   STATUS[148].EXT.Operation := FALSE;
   STATUS[148].EXT.Forced := FALSE;
   STATUS[148].EXT.BIT29 := FALSE;
   STATUS[148].EXT.BIT30 := FALSE;
   STATUS[148].EXT.BIT31 := FALSE;
   STATUS[148].EXT.ModeBit1 := FALSE;
   STATUS[148].EXT.ModeBit2 := FALSE;
   STATUS[148].EXT.ModeBit3 := FALSE;
   STATUS[148].EXT.BIT19 := FALSE;
   STATUS[148].EXT.BIT20 := FALSE;
   STATUS[148].EXT.AlarmSuppressed := FALSE;
   STATUS[148].EXT.AlarmPresent := FALSE;
   STATUS[148].EXT.AlarmFailUnAck := FALSE;
   STATUS[148].Status := 0;
   STATUS[148].TimeStamp := 16#0000;
   STATUS[149].EXT.AlarmWarnUnAck := FALSE;
   STATUS[149].EXT.AckRequired := FALSE;
   STATUS[149].EXT.Maintanence := FALSE;
   STATUS[149].EXT.Operation := FALSE;
   STATUS[149].EXT.Forced := FALSE;
   STATUS[149].EXT.BIT29 := FALSE;
   STATUS[149].EXT.BIT30 := FALSE;
   STATUS[149].EXT.BIT31 := FALSE;
   STATUS[149].EXT.ModeBit1 := FALSE;
   STATUS[149].EXT.ModeBit2 := FALSE;
   STATUS[149].EXT.ModeBit3 := FALSE;
   STATUS[149].EXT.BIT19 := FALSE;
   STATUS[149].EXT.BIT20 := FALSE;
   STATUS[149].EXT.AlarmSuppressed := FALSE;
   STATUS[149].EXT.AlarmPresent := FALSE;
   STATUS[149].EXT.AlarmFailUnAck := FALSE;
   STATUS[149].Status := 0;
   STATUS[149].TimeStamp := 16#0000;
   STATUS[150].EXT.AlarmWarnUnAck := FALSE;
   STATUS[150].EXT.AckRequired := FALSE;
   STATUS[150].EXT.Maintanence := FALSE;
   STATUS[150].EXT.Operation := FALSE;
   STATUS[150].EXT.Forced := FALSE;
   STATUS[150].EXT.BIT29 := FALSE;
   STATUS[150].EXT.BIT30 := FALSE;
   STATUS[150].EXT.BIT31 := FALSE;
   STATUS[150].EXT.ModeBit1 := FALSE;
   STATUS[150].EXT.ModeBit2 := FALSE;
   STATUS[150].EXT.ModeBit3 := FALSE;
   STATUS[150].EXT.BIT19 := FALSE;
   STATUS[150].EXT.BIT20 := FALSE;
   STATUS[150].EXT.AlarmSuppressed := FALSE;
   STATUS[150].EXT.AlarmPresent := FALSE;
   STATUS[150].EXT.AlarmFailUnAck := FALSE;
   STATUS[150].Status := 0;
   STATUS[150].TimeStamp := 16#0000;
   STATUS[151].EXT.AlarmWarnUnAck := FALSE;
   STATUS[151].EXT.AckRequired := FALSE;
   STATUS[151].EXT.Maintanence := FALSE;
   STATUS[151].EXT.Operation := FALSE;
   STATUS[151].EXT.Forced := FALSE;
   STATUS[151].EXT.BIT29 := FALSE;
   STATUS[151].EXT.BIT30 := FALSE;
   STATUS[151].EXT.BIT31 := FALSE;
   STATUS[151].EXT.ModeBit1 := FALSE;
   STATUS[151].EXT.ModeBit2 := FALSE;
   STATUS[151].EXT.ModeBit3 := FALSE;
   STATUS[151].EXT.BIT19 := FALSE;
   STATUS[151].EXT.BIT20 := FALSE;
   STATUS[151].EXT.AlarmSuppressed := FALSE;
   STATUS[151].EXT.AlarmPresent := FALSE;
   STATUS[151].EXT.AlarmFailUnAck := FALSE;
   STATUS[151].Status := 0;
   STATUS[151].TimeStamp := 16#0000;
   STATUS[152].EXT.AlarmWarnUnAck := FALSE;
   STATUS[152].EXT.AckRequired := FALSE;
   STATUS[152].EXT.Maintanence := FALSE;
   STATUS[152].EXT.Operation := FALSE;
   STATUS[152].EXT.Forced := FALSE;
   STATUS[152].EXT.BIT29 := FALSE;
   STATUS[152].EXT.BIT30 := FALSE;
   STATUS[152].EXT.BIT31 := FALSE;
   STATUS[152].EXT.ModeBit1 := FALSE;
   STATUS[152].EXT.ModeBit2 := FALSE;
   STATUS[152].EXT.ModeBit3 := FALSE;
   STATUS[152].EXT.BIT19 := FALSE;
   STATUS[152].EXT.BIT20 := FALSE;
   STATUS[152].EXT.AlarmSuppressed := FALSE;
   STATUS[152].EXT.AlarmPresent := FALSE;
   STATUS[152].EXT.AlarmFailUnAck := FALSE;
   STATUS[152].Status := 0;
   STATUS[152].TimeStamp := 16#0000;
   STATUS[153].EXT.AlarmWarnUnAck := FALSE;
   STATUS[153].EXT.AckRequired := FALSE;
   STATUS[153].EXT.Maintanence := FALSE;
   STATUS[153].EXT.Operation := FALSE;
   STATUS[153].EXT.Forced := FALSE;
   STATUS[153].EXT.BIT29 := FALSE;
   STATUS[153].EXT.BIT30 := FALSE;
   STATUS[153].EXT.BIT31 := FALSE;
   STATUS[153].EXT.ModeBit1 := FALSE;
   STATUS[153].EXT.ModeBit2 := FALSE;
   STATUS[153].EXT.ModeBit3 := FALSE;
   STATUS[153].EXT.BIT19 := FALSE;
   STATUS[153].EXT.BIT20 := FALSE;
   STATUS[153].EXT.AlarmSuppressed := FALSE;
   STATUS[153].EXT.AlarmPresent := FALSE;
   STATUS[153].EXT.AlarmFailUnAck := FALSE;
   STATUS[153].Status := 0;
   STATUS[153].TimeStamp := 16#0000;
   STATUS[154].EXT.AlarmWarnUnAck := FALSE;
   STATUS[154].EXT.AckRequired := FALSE;
   STATUS[154].EXT.Maintanence := FALSE;
   STATUS[154].EXT.Operation := FALSE;
   STATUS[154].EXT.Forced := FALSE;
   STATUS[154].EXT.BIT29 := FALSE;
   STATUS[154].EXT.BIT30 := FALSE;
   STATUS[154].EXT.BIT31 := FALSE;
   STATUS[154].EXT.ModeBit1 := FALSE;
   STATUS[154].EXT.ModeBit2 := FALSE;
   STATUS[154].EXT.ModeBit3 := FALSE;
   STATUS[154].EXT.BIT19 := FALSE;
   STATUS[154].EXT.BIT20 := FALSE;
   STATUS[154].EXT.AlarmSuppressed := FALSE;
   STATUS[154].EXT.AlarmPresent := FALSE;
   STATUS[154].EXT.AlarmFailUnAck := FALSE;
   STATUS[154].Status := 0;
   STATUS[154].TimeStamp := 16#0000;
   STATUS[155].EXT.AlarmWarnUnAck := FALSE;
   STATUS[155].EXT.AckRequired := FALSE;
   STATUS[155].EXT.Maintanence := FALSE;
   STATUS[155].EXT.Operation := FALSE;
   STATUS[155].EXT.Forced := FALSE;
   STATUS[155].EXT.BIT29 := FALSE;
   STATUS[155].EXT.BIT30 := FALSE;
   STATUS[155].EXT.BIT31 := FALSE;
   STATUS[155].EXT.ModeBit1 := FALSE;
   STATUS[155].EXT.ModeBit2 := FALSE;
   STATUS[155].EXT.ModeBit3 := FALSE;
   STATUS[155].EXT.BIT19 := FALSE;
   STATUS[155].EXT.BIT20 := FALSE;
   STATUS[155].EXT.AlarmSuppressed := FALSE;
   STATUS[155].EXT.AlarmPresent := FALSE;
   STATUS[155].EXT.AlarmFailUnAck := FALSE;
   STATUS[155].Status := 0;
   STATUS[155].TimeStamp := 16#0000;
   STATUS[156].EXT.AlarmWarnUnAck := FALSE;
   STATUS[156].EXT.AckRequired := FALSE;
   STATUS[156].EXT.Maintanence := FALSE;
   STATUS[156].EXT.Operation := FALSE;
   STATUS[156].EXT.Forced := FALSE;
   STATUS[156].EXT.BIT29 := FALSE;
   STATUS[156].EXT.BIT30 := FALSE;
   STATUS[156].EXT.BIT31 := FALSE;
   STATUS[156].EXT.ModeBit1 := FALSE;
   STATUS[156].EXT.ModeBit2 := FALSE;
   STATUS[156].EXT.ModeBit3 := FALSE;
   STATUS[156].EXT.BIT19 := FALSE;
   STATUS[156].EXT.BIT20 := FALSE;
   STATUS[156].EXT.AlarmSuppressed := FALSE;
   STATUS[156].EXT.AlarmPresent := FALSE;
   STATUS[156].EXT.AlarmFailUnAck := FALSE;
   STATUS[156].Status := 0;
   STATUS[156].TimeStamp := 16#0000;
   STATUS[157].EXT.AlarmWarnUnAck := FALSE;
   STATUS[157].EXT.AckRequired := FALSE;
   STATUS[157].EXT.Maintanence := FALSE;
   STATUS[157].EXT.Operation := FALSE;
   STATUS[157].EXT.Forced := FALSE;
   STATUS[157].EXT.BIT29 := FALSE;
   STATUS[157].EXT.BIT30 := FALSE;
   STATUS[157].EXT.BIT31 := FALSE;
   STATUS[157].EXT.ModeBit1 := FALSE;
   STATUS[157].EXT.ModeBit2 := FALSE;
   STATUS[157].EXT.ModeBit3 := FALSE;
   STATUS[157].EXT.BIT19 := FALSE;
   STATUS[157].EXT.BIT20 := FALSE;
   STATUS[157].EXT.AlarmSuppressed := FALSE;
   STATUS[157].EXT.AlarmPresent := FALSE;
   STATUS[157].EXT.AlarmFailUnAck := FALSE;
   STATUS[157].Status := 0;
   STATUS[157].TimeStamp := 16#0000;
   STATUS[158].EXT.AlarmWarnUnAck := FALSE;
   STATUS[158].EXT.AckRequired := FALSE;
   STATUS[158].EXT.Maintanence := FALSE;
   STATUS[158].EXT.Operation := FALSE;
   STATUS[158].EXT.Forced := FALSE;
   STATUS[158].EXT.BIT29 := FALSE;
   STATUS[158].EXT.BIT30 := FALSE;
   STATUS[158].EXT.BIT31 := FALSE;
   STATUS[158].EXT.ModeBit1 := FALSE;
   STATUS[158].EXT.ModeBit2 := FALSE;
   STATUS[158].EXT.ModeBit3 := FALSE;
   STATUS[158].EXT.BIT19 := FALSE;
   STATUS[158].EXT.BIT20 := FALSE;
   STATUS[158].EXT.AlarmSuppressed := FALSE;
   STATUS[158].EXT.AlarmPresent := FALSE;
   STATUS[158].EXT.AlarmFailUnAck := FALSE;
   STATUS[158].Status := 0;
   STATUS[158].TimeStamp := 16#0000;
   STATUS[159].EXT.AlarmWarnUnAck := FALSE;
   STATUS[159].EXT.AckRequired := FALSE;
   STATUS[159].EXT.Maintanence := FALSE;
   STATUS[159].EXT.Operation := FALSE;
   STATUS[159].EXT.Forced := FALSE;
   STATUS[159].EXT.BIT29 := FALSE;
   STATUS[159].EXT.BIT30 := FALSE;
   STATUS[159].EXT.BIT31 := FALSE;
   STATUS[159].EXT.ModeBit1 := FALSE;
   STATUS[159].EXT.ModeBit2 := FALSE;
   STATUS[159].EXT.ModeBit3 := FALSE;
   STATUS[159].EXT.BIT19 := FALSE;
   STATUS[159].EXT.BIT20 := FALSE;
   STATUS[159].EXT.AlarmSuppressed := FALSE;
   STATUS[159].EXT.AlarmPresent := FALSE;
   STATUS[159].EXT.AlarmFailUnAck := FALSE;
   STATUS[159].Status := 0;
   STATUS[159].TimeStamp := 16#0000;
   STATUS[160].EXT.AlarmWarnUnAck := FALSE;
   STATUS[160].EXT.AckRequired := FALSE;
   STATUS[160].EXT.Maintanence := FALSE;
   STATUS[160].EXT.Operation := FALSE;
   STATUS[160].EXT.Forced := FALSE;
   STATUS[160].EXT.BIT29 := FALSE;
   STATUS[160].EXT.BIT30 := FALSE;
   STATUS[160].EXT.BIT31 := FALSE;
   STATUS[160].EXT.ModeBit1 := FALSE;
   STATUS[160].EXT.ModeBit2 := FALSE;
   STATUS[160].EXT.ModeBit3 := FALSE;
   STATUS[160].EXT.BIT19 := FALSE;
   STATUS[160].EXT.BIT20 := FALSE;
   STATUS[160].EXT.AlarmSuppressed := FALSE;
   STATUS[160].EXT.AlarmPresent := FALSE;
   STATUS[160].EXT.AlarmFailUnAck := FALSE;
   STATUS[160].Status := 0;
   STATUS[160].TimeStamp := 16#0000;
   STATUS[161].EXT.AlarmWarnUnAck := FALSE;
   STATUS[161].EXT.AckRequired := FALSE;
   STATUS[161].EXT.Maintanence := FALSE;
   STATUS[161].EXT.Operation := FALSE;
   STATUS[161].EXT.Forced := FALSE;
   STATUS[161].EXT.BIT29 := FALSE;
   STATUS[161].EXT.BIT30 := FALSE;
   STATUS[161].EXT.BIT31 := FALSE;
   STATUS[161].EXT.ModeBit1 := FALSE;
   STATUS[161].EXT.ModeBit2 := FALSE;
   STATUS[161].EXT.ModeBit3 := FALSE;
   STATUS[161].EXT.BIT19 := FALSE;
   STATUS[161].EXT.BIT20 := FALSE;
   STATUS[161].EXT.AlarmSuppressed := FALSE;
   STATUS[161].EXT.AlarmPresent := FALSE;
   STATUS[161].EXT.AlarmFailUnAck := FALSE;
   STATUS[161].Status := 0;
   STATUS[161].TimeStamp := 16#0000;
   STATUS[162].EXT.AlarmWarnUnAck := FALSE;
   STATUS[162].EXT.AckRequired := FALSE;
   STATUS[162].EXT.Maintanence := FALSE;
   STATUS[162].EXT.Operation := FALSE;
   STATUS[162].EXT.Forced := FALSE;
   STATUS[162].EXT.BIT29 := FALSE;
   STATUS[162].EXT.BIT30 := FALSE;
   STATUS[162].EXT.BIT31 := FALSE;
   STATUS[162].EXT.ModeBit1 := FALSE;
   STATUS[162].EXT.ModeBit2 := FALSE;
   STATUS[162].EXT.ModeBit3 := FALSE;
   STATUS[162].EXT.BIT19 := FALSE;
   STATUS[162].EXT.BIT20 := FALSE;
   STATUS[162].EXT.AlarmSuppressed := FALSE;
   STATUS[162].EXT.AlarmPresent := FALSE;
   STATUS[162].EXT.AlarmFailUnAck := FALSE;
   STATUS[162].Status := 0;
   STATUS[162].TimeStamp := 16#0000;
   STATUS[163].EXT.AlarmWarnUnAck := FALSE;
   STATUS[163].EXT.AckRequired := FALSE;
   STATUS[163].EXT.Maintanence := FALSE;
   STATUS[163].EXT.Operation := FALSE;
   STATUS[163].EXT.Forced := FALSE;
   STATUS[163].EXT.BIT29 := FALSE;
   STATUS[163].EXT.BIT30 := FALSE;
   STATUS[163].EXT.BIT31 := FALSE;
   STATUS[163].EXT.ModeBit1 := FALSE;
   STATUS[163].EXT.ModeBit2 := FALSE;
   STATUS[163].EXT.ModeBit3 := FALSE;
   STATUS[163].EXT.BIT19 := FALSE;
   STATUS[163].EXT.BIT20 := FALSE;
   STATUS[163].EXT.AlarmSuppressed := FALSE;
   STATUS[163].EXT.AlarmPresent := FALSE;
   STATUS[163].EXT.AlarmFailUnAck := FALSE;
   STATUS[163].Status := 0;
   STATUS[163].TimeStamp := 16#0000;
   STATUS[164].EXT.AlarmWarnUnAck := FALSE;
   STATUS[164].EXT.AckRequired := FALSE;
   STATUS[164].EXT.Maintanence := FALSE;
   STATUS[164].EXT.Operation := FALSE;
   STATUS[164].EXT.Forced := FALSE;
   STATUS[164].EXT.BIT29 := FALSE;
   STATUS[164].EXT.BIT30 := FALSE;
   STATUS[164].EXT.BIT31 := FALSE;
   STATUS[164].EXT.ModeBit1 := FALSE;
   STATUS[164].EXT.ModeBit2 := FALSE;
   STATUS[164].EXT.ModeBit3 := FALSE;
   STATUS[164].EXT.BIT19 := FALSE;
   STATUS[164].EXT.BIT20 := FALSE;
   STATUS[164].EXT.AlarmSuppressed := FALSE;
   STATUS[164].EXT.AlarmPresent := FALSE;
   STATUS[164].EXT.AlarmFailUnAck := FALSE;
   STATUS[164].Status := 0;
   STATUS[164].TimeStamp := 16#0000;
   STATUS[165].EXT.AlarmWarnUnAck := FALSE;
   STATUS[165].EXT.AckRequired := FALSE;
   STATUS[165].EXT.Maintanence := FALSE;
   STATUS[165].EXT.Operation := FALSE;
   STATUS[165].EXT.Forced := FALSE;
   STATUS[165].EXT.BIT29 := FALSE;
   STATUS[165].EXT.BIT30 := FALSE;
   STATUS[165].EXT.BIT31 := FALSE;
   STATUS[165].EXT.ModeBit1 := FALSE;
   STATUS[165].EXT.ModeBit2 := FALSE;
   STATUS[165].EXT.ModeBit3 := FALSE;
   STATUS[165].EXT.BIT19 := FALSE;
   STATUS[165].EXT.BIT20 := FALSE;
   STATUS[165].EXT.AlarmSuppressed := FALSE;
   STATUS[165].EXT.AlarmPresent := FALSE;
   STATUS[165].EXT.AlarmFailUnAck := FALSE;
   STATUS[165].Status := 0;
   STATUS[165].TimeStamp := 16#0000;
   STATUS[166].EXT.AlarmWarnUnAck := FALSE;
   STATUS[166].EXT.AckRequired := FALSE;
   STATUS[166].EXT.Maintanence := FALSE;
   STATUS[166].EXT.Operation := FALSE;
   STATUS[166].EXT.Forced := FALSE;
   STATUS[166].EXT.BIT29 := FALSE;
   STATUS[166].EXT.BIT30 := FALSE;
   STATUS[166].EXT.BIT31 := FALSE;
   STATUS[166].EXT.ModeBit1 := FALSE;
   STATUS[166].EXT.ModeBit2 := FALSE;
   STATUS[166].EXT.ModeBit3 := FALSE;
   STATUS[166].EXT.BIT19 := FALSE;
   STATUS[166].EXT.BIT20 := FALSE;
   STATUS[166].EXT.AlarmSuppressed := FALSE;
   STATUS[166].EXT.AlarmPresent := FALSE;
   STATUS[166].EXT.AlarmFailUnAck := FALSE;
   STATUS[166].Status := 0;
   STATUS[166].TimeStamp := 16#0000;
   STATUS[167].EXT.AlarmWarnUnAck := FALSE;
   STATUS[167].EXT.AckRequired := FALSE;
   STATUS[167].EXT.Maintanence := FALSE;
   STATUS[167].EXT.Operation := FALSE;
   STATUS[167].EXT.Forced := FALSE;
   STATUS[167].EXT.BIT29 := FALSE;
   STATUS[167].EXT.BIT30 := FALSE;
   STATUS[167].EXT.BIT31 := FALSE;
   STATUS[167].EXT.ModeBit1 := FALSE;
   STATUS[167].EXT.ModeBit2 := FALSE;
   STATUS[167].EXT.ModeBit3 := FALSE;
   STATUS[167].EXT.BIT19 := FALSE;
   STATUS[167].EXT.BIT20 := FALSE;
   STATUS[167].EXT.AlarmSuppressed := FALSE;
   STATUS[167].EXT.AlarmPresent := FALSE;
   STATUS[167].EXT.AlarmFailUnAck := FALSE;
   STATUS[167].Status := 0;
   STATUS[167].TimeStamp := 16#0000;
   STATUS[168].EXT.AlarmWarnUnAck := FALSE;
   STATUS[168].EXT.AckRequired := FALSE;
   STATUS[168].EXT.Maintanence := FALSE;
   STATUS[168].EXT.Operation := FALSE;
   STATUS[168].EXT.Forced := FALSE;
   STATUS[168].EXT.BIT29 := FALSE;
   STATUS[168].EXT.BIT30 := FALSE;
   STATUS[168].EXT.BIT31 := FALSE;
   STATUS[168].EXT.ModeBit1 := FALSE;
   STATUS[168].EXT.ModeBit2 := FALSE;
   STATUS[168].EXT.ModeBit3 := FALSE;
   STATUS[168].EXT.BIT19 := FALSE;
   STATUS[168].EXT.BIT20 := FALSE;
   STATUS[168].EXT.AlarmSuppressed := FALSE;
   STATUS[168].EXT.AlarmPresent := FALSE;
   STATUS[168].EXT.AlarmFailUnAck := FALSE;
   STATUS[168].Status := 0;
   STATUS[168].TimeStamp := 16#0000;
   STATUS[169].EXT.AlarmWarnUnAck := FALSE;
   STATUS[169].EXT.AckRequired := FALSE;
   STATUS[169].EXT.Maintanence := FALSE;
   STATUS[169].EXT.Operation := FALSE;
   STATUS[169].EXT.Forced := FALSE;
   STATUS[169].EXT.BIT29 := FALSE;
   STATUS[169].EXT.BIT30 := FALSE;
   STATUS[169].EXT.BIT31 := FALSE;
   STATUS[169].EXT.ModeBit1 := FALSE;
   STATUS[169].EXT.ModeBit2 := FALSE;
   STATUS[169].EXT.ModeBit3 := FALSE;
   STATUS[169].EXT.BIT19 := FALSE;
   STATUS[169].EXT.BIT20 := FALSE;
   STATUS[169].EXT.AlarmSuppressed := FALSE;
   STATUS[169].EXT.AlarmPresent := FALSE;
   STATUS[169].EXT.AlarmFailUnAck := FALSE;
   STATUS[169].Status := 0;
   STATUS[169].TimeStamp := 16#0000;
   STATUS[170].EXT.AlarmWarnUnAck := FALSE;
   STATUS[170].EXT.AckRequired := FALSE;
   STATUS[170].EXT.Maintanence := FALSE;
   STATUS[170].EXT.Operation := FALSE;
   STATUS[170].EXT.Forced := FALSE;
   STATUS[170].EXT.BIT29 := FALSE;
   STATUS[170].EXT.BIT30 := FALSE;
   STATUS[170].EXT.BIT31 := FALSE;
   STATUS[170].EXT.ModeBit1 := FALSE;
   STATUS[170].EXT.ModeBit2 := FALSE;
   STATUS[170].EXT.ModeBit3 := FALSE;
   STATUS[170].EXT.BIT19 := FALSE;
   STATUS[170].EXT.BIT20 := FALSE;
   STATUS[170].EXT.AlarmSuppressed := FALSE;
   STATUS[170].EXT.AlarmPresent := FALSE;
   STATUS[170].EXT.AlarmFailUnAck := FALSE;
   STATUS[170].Status := 0;
   STATUS[170].TimeStamp := 16#0000;
   STATUS[171].EXT.AlarmWarnUnAck := FALSE;
   STATUS[171].EXT.AckRequired := FALSE;
   STATUS[171].EXT.Maintanence := FALSE;
   STATUS[171].EXT.Operation := FALSE;
   STATUS[171].EXT.Forced := FALSE;
   STATUS[171].EXT.BIT29 := FALSE;
   STATUS[171].EXT.BIT30 := FALSE;
   STATUS[171].EXT.BIT31 := FALSE;
   STATUS[171].EXT.ModeBit1 := FALSE;
   STATUS[171].EXT.ModeBit2 := FALSE;
   STATUS[171].EXT.ModeBit3 := FALSE;
   STATUS[171].EXT.BIT19 := FALSE;
   STATUS[171].EXT.BIT20 := FALSE;
   STATUS[171].EXT.AlarmSuppressed := FALSE;
   STATUS[171].EXT.AlarmPresent := FALSE;
   STATUS[171].EXT.AlarmFailUnAck := FALSE;
   STATUS[171].Status := 0;
   STATUS[171].TimeStamp := 16#0000;
   STATUS[172].EXT.AlarmWarnUnAck := FALSE;
   STATUS[172].EXT.AckRequired := FALSE;
   STATUS[172].EXT.Maintanence := FALSE;
   STATUS[172].EXT.Operation := FALSE;
   STATUS[172].EXT.Forced := FALSE;
   STATUS[172].EXT.BIT29 := FALSE;
   STATUS[172].EXT.BIT30 := FALSE;
   STATUS[172].EXT.BIT31 := FALSE;
   STATUS[172].EXT.ModeBit1 := FALSE;
   STATUS[172].EXT.ModeBit2 := FALSE;
   STATUS[172].EXT.ModeBit3 := FALSE;
   STATUS[172].EXT.BIT19 := FALSE;
   STATUS[172].EXT.BIT20 := FALSE;
   STATUS[172].EXT.AlarmSuppressed := FALSE;
   STATUS[172].EXT.AlarmPresent := FALSE;
   STATUS[172].EXT.AlarmFailUnAck := FALSE;
   STATUS[172].Status := 0;
   STATUS[172].TimeStamp := 16#0000;
   STATUS[173].EXT.AlarmWarnUnAck := FALSE;
   STATUS[173].EXT.AckRequired := FALSE;
   STATUS[173].EXT.Maintanence := FALSE;
   STATUS[173].EXT.Operation := FALSE;
   STATUS[173].EXT.Forced := FALSE;
   STATUS[173].EXT.BIT29 := FALSE;
   STATUS[173].EXT.BIT30 := FALSE;
   STATUS[173].EXT.BIT31 := FALSE;
   STATUS[173].EXT.ModeBit1 := FALSE;
   STATUS[173].EXT.ModeBit2 := FALSE;
   STATUS[173].EXT.ModeBit3 := FALSE;
   STATUS[173].EXT.BIT19 := FALSE;
   STATUS[173].EXT.BIT20 := FALSE;
   STATUS[173].EXT.AlarmSuppressed := FALSE;
   STATUS[173].EXT.AlarmPresent := FALSE;
   STATUS[173].EXT.AlarmFailUnAck := FALSE;
   STATUS[173].Status := 0;
   STATUS[173].TimeStamp := 16#0000;
   STATUS[174].EXT.AlarmWarnUnAck := FALSE;
   STATUS[174].EXT.AckRequired := FALSE;
   STATUS[174].EXT.Maintanence := FALSE;
   STATUS[174].EXT.Operation := FALSE;
   STATUS[174].EXT.Forced := FALSE;
   STATUS[174].EXT.BIT29 := FALSE;
   STATUS[174].EXT.BIT30 := FALSE;
   STATUS[174].EXT.BIT31 := FALSE;
   STATUS[174].EXT.ModeBit1 := FALSE;
   STATUS[174].EXT.ModeBit2 := FALSE;
   STATUS[174].EXT.ModeBit3 := FALSE;
   STATUS[174].EXT.BIT19 := FALSE;
   STATUS[174].EXT.BIT20 := FALSE;
   STATUS[174].EXT.AlarmSuppressed := FALSE;
   STATUS[174].EXT.AlarmPresent := FALSE;
   STATUS[174].EXT.AlarmFailUnAck := FALSE;
   STATUS[174].Status := 0;
   STATUS[174].TimeStamp := 16#0000;
   STATUS[175].EXT.AlarmWarnUnAck := FALSE;
   STATUS[175].EXT.AckRequired := FALSE;
   STATUS[175].EXT.Maintanence := FALSE;
   STATUS[175].EXT.Operation := FALSE;
   STATUS[175].EXT.Forced := FALSE;
   STATUS[175].EXT.BIT29 := FALSE;
   STATUS[175].EXT.BIT30 := FALSE;
   STATUS[175].EXT.BIT31 := FALSE;
   STATUS[175].EXT.ModeBit1 := FALSE;
   STATUS[175].EXT.ModeBit2 := FALSE;
   STATUS[175].EXT.ModeBit3 := FALSE;
   STATUS[175].EXT.BIT19 := FALSE;
   STATUS[175].EXT.BIT20 := FALSE;
   STATUS[175].EXT.AlarmSuppressed := FALSE;
   STATUS[175].EXT.AlarmPresent := FALSE;
   STATUS[175].EXT.AlarmFailUnAck := FALSE;
   STATUS[175].Status := 0;
   STATUS[175].TimeStamp := 16#0000;
   STATUS[176].EXT.AlarmWarnUnAck := FALSE;
   STATUS[176].EXT.AckRequired := FALSE;
   STATUS[176].EXT.Maintanence := FALSE;
   STATUS[176].EXT.Operation := FALSE;
   STATUS[176].EXT.Forced := FALSE;
   STATUS[176].EXT.BIT29 := FALSE;
   STATUS[176].EXT.BIT30 := FALSE;
   STATUS[176].EXT.BIT31 := FALSE;
   STATUS[176].EXT.ModeBit1 := FALSE;
   STATUS[176].EXT.ModeBit2 := FALSE;
   STATUS[176].EXT.ModeBit3 := FALSE;
   STATUS[176].EXT.BIT19 := FALSE;
   STATUS[176].EXT.BIT20 := FALSE;
   STATUS[176].EXT.AlarmSuppressed := FALSE;
   STATUS[176].EXT.AlarmPresent := FALSE;
   STATUS[176].EXT.AlarmFailUnAck := FALSE;
   STATUS[176].Status := 0;
   STATUS[176].TimeStamp := 16#0000;
   STATUS[177].EXT.AlarmWarnUnAck := FALSE;
   STATUS[177].EXT.AckRequired := FALSE;
   STATUS[177].EXT.Maintanence := FALSE;
   STATUS[177].EXT.Operation := FALSE;
   STATUS[177].EXT.Forced := FALSE;
   STATUS[177].EXT.BIT29 := FALSE;
   STATUS[177].EXT.BIT30 := FALSE;
   STATUS[177].EXT.BIT31 := FALSE;
   STATUS[177].EXT.ModeBit1 := FALSE;
   STATUS[177].EXT.ModeBit2 := FALSE;
   STATUS[177].EXT.ModeBit3 := FALSE;
   STATUS[177].EXT.BIT19 := FALSE;
   STATUS[177].EXT.BIT20 := FALSE;
   STATUS[177].EXT.AlarmSuppressed := FALSE;
   STATUS[177].EXT.AlarmPresent := FALSE;
   STATUS[177].EXT.AlarmFailUnAck := FALSE;
   STATUS[177].Status := 0;
   STATUS[177].TimeStamp := 16#0000;
   STATUS[178].EXT.AlarmWarnUnAck := FALSE;
   STATUS[178].EXT.AckRequired := FALSE;
   STATUS[178].EXT.Maintanence := FALSE;
   STATUS[178].EXT.Operation := FALSE;
   STATUS[178].EXT.Forced := FALSE;
   STATUS[178].EXT.BIT29 := FALSE;
   STATUS[178].EXT.BIT30 := FALSE;
   STATUS[178].EXT.BIT31 := FALSE;
   STATUS[178].EXT.ModeBit1 := FALSE;
   STATUS[178].EXT.ModeBit2 := FALSE;
   STATUS[178].EXT.ModeBit3 := FALSE;
   STATUS[178].EXT.BIT19 := FALSE;
   STATUS[178].EXT.BIT20 := FALSE;
   STATUS[178].EXT.AlarmSuppressed := FALSE;
   STATUS[178].EXT.AlarmPresent := FALSE;
   STATUS[178].EXT.AlarmFailUnAck := FALSE;
   STATUS[178].Status := 0;
   STATUS[178].TimeStamp := 16#0000;
   STATUS[179].EXT.AlarmWarnUnAck := FALSE;
   STATUS[179].EXT.AckRequired := FALSE;
   STATUS[179].EXT.Maintanence := FALSE;
   STATUS[179].EXT.Operation := FALSE;
   STATUS[179].EXT.Forced := FALSE;
   STATUS[179].EXT.BIT29 := FALSE;
   STATUS[179].EXT.BIT30 := FALSE;
   STATUS[179].EXT.BIT31 := FALSE;
   STATUS[179].EXT.ModeBit1 := FALSE;
   STATUS[179].EXT.ModeBit2 := FALSE;
   STATUS[179].EXT.ModeBit3 := FALSE;
   STATUS[179].EXT.BIT19 := FALSE;
   STATUS[179].EXT.BIT20 := FALSE;
   STATUS[179].EXT.AlarmSuppressed := FALSE;
   STATUS[179].EXT.AlarmPresent := FALSE;
   STATUS[179].EXT.AlarmFailUnAck := FALSE;
   STATUS[179].Status := 0;
   STATUS[179].TimeStamp := 16#0000;
   STATUS[180].EXT.AlarmWarnUnAck := FALSE;
   STATUS[180].EXT.AckRequired := FALSE;
   STATUS[180].EXT.Maintanence := FALSE;
   STATUS[180].EXT.Operation := FALSE;
   STATUS[180].EXT.Forced := FALSE;
   STATUS[180].EXT.BIT29 := FALSE;
   STATUS[180].EXT.BIT30 := FALSE;
   STATUS[180].EXT.BIT31 := FALSE;
   STATUS[180].EXT.ModeBit1 := FALSE;
   STATUS[180].EXT.ModeBit2 := FALSE;
   STATUS[180].EXT.ModeBit3 := FALSE;
   STATUS[180].EXT.BIT19 := FALSE;
   STATUS[180].EXT.BIT20 := FALSE;
   STATUS[180].EXT.AlarmSuppressed := FALSE;
   STATUS[180].EXT.AlarmPresent := FALSE;
   STATUS[180].EXT.AlarmFailUnAck := FALSE;
   STATUS[180].Status := 0;
   STATUS[180].TimeStamp := 16#0000;
   STATUS[181].EXT.AlarmWarnUnAck := FALSE;
   STATUS[181].EXT.AckRequired := FALSE;
   STATUS[181].EXT.Maintanence := FALSE;
   STATUS[181].EXT.Operation := FALSE;
   STATUS[181].EXT.Forced := FALSE;
   STATUS[181].EXT.BIT29 := FALSE;
   STATUS[181].EXT.BIT30 := FALSE;
   STATUS[181].EXT.BIT31 := FALSE;
   STATUS[181].EXT.ModeBit1 := FALSE;
   STATUS[181].EXT.ModeBit2 := FALSE;
   STATUS[181].EXT.ModeBit3 := FALSE;
   STATUS[181].EXT.BIT19 := FALSE;
   STATUS[181].EXT.BIT20 := FALSE;
   STATUS[181].EXT.AlarmSuppressed := FALSE;
   STATUS[181].EXT.AlarmPresent := FALSE;
   STATUS[181].EXT.AlarmFailUnAck := FALSE;
   STATUS[181].Status := 0;
   STATUS[181].TimeStamp := 16#0000;
   STATUS[182].EXT.AlarmWarnUnAck := FALSE;
   STATUS[182].EXT.AckRequired := FALSE;
   STATUS[182].EXT.Maintanence := FALSE;
   STATUS[182].EXT.Operation := FALSE;
   STATUS[182].EXT.Forced := FALSE;
   STATUS[182].EXT.BIT29 := FALSE;
   STATUS[182].EXT.BIT30 := FALSE;
   STATUS[182].EXT.BIT31 := FALSE;
   STATUS[182].EXT.ModeBit1 := FALSE;
   STATUS[182].EXT.ModeBit2 := FALSE;
   STATUS[182].EXT.ModeBit3 := FALSE;
   STATUS[182].EXT.BIT19 := FALSE;
   STATUS[182].EXT.BIT20 := FALSE;
   STATUS[182].EXT.AlarmSuppressed := FALSE;
   STATUS[182].EXT.AlarmPresent := FALSE;
   STATUS[182].EXT.AlarmFailUnAck := FALSE;
   STATUS[182].Status := 0;
   STATUS[182].TimeStamp := 16#0000;
   STATUS[183].EXT.AlarmWarnUnAck := FALSE;
   STATUS[183].EXT.AckRequired := FALSE;
   STATUS[183].EXT.Maintanence := FALSE;
   STATUS[183].EXT.Operation := FALSE;
   STATUS[183].EXT.Forced := FALSE;
   STATUS[183].EXT.BIT29 := FALSE;
   STATUS[183].EXT.BIT30 := FALSE;
   STATUS[183].EXT.BIT31 := FALSE;
   STATUS[183].EXT.ModeBit1 := FALSE;
   STATUS[183].EXT.ModeBit2 := FALSE;
   STATUS[183].EXT.ModeBit3 := FALSE;
   STATUS[183].EXT.BIT19 := FALSE;
   STATUS[183].EXT.BIT20 := FALSE;
   STATUS[183].EXT.AlarmSuppressed := FALSE;
   STATUS[183].EXT.AlarmPresent := FALSE;
   STATUS[183].EXT.AlarmFailUnAck := FALSE;
   STATUS[183].Status := 0;
   STATUS[183].TimeStamp := 16#0000;
   STATUS[184].EXT.AlarmWarnUnAck := FALSE;
   STATUS[184].EXT.AckRequired := FALSE;
   STATUS[184].EXT.Maintanence := FALSE;
   STATUS[184].EXT.Operation := FALSE;
   STATUS[184].EXT.Forced := FALSE;
   STATUS[184].EXT.BIT29 := FALSE;
   STATUS[184].EXT.BIT30 := FALSE;
   STATUS[184].EXT.BIT31 := FALSE;
   STATUS[184].EXT.ModeBit1 := FALSE;
   STATUS[184].EXT.ModeBit2 := FALSE;
   STATUS[184].EXT.ModeBit3 := FALSE;
   STATUS[184].EXT.BIT19 := FALSE;
   STATUS[184].EXT.BIT20 := FALSE;
   STATUS[184].EXT.AlarmSuppressed := FALSE;
   STATUS[184].EXT.AlarmPresent := FALSE;
   STATUS[184].EXT.AlarmFailUnAck := FALSE;
   STATUS[184].Status := 0;
   STATUS[184].TimeStamp := 16#0000;
   STATUS[185].EXT.AlarmWarnUnAck := FALSE;
   STATUS[185].EXT.AckRequired := FALSE;
   STATUS[185].EXT.Maintanence := FALSE;
   STATUS[185].EXT.Operation := FALSE;
   STATUS[185].EXT.Forced := FALSE;
   STATUS[185].EXT.BIT29 := FALSE;
   STATUS[185].EXT.BIT30 := FALSE;
   STATUS[185].EXT.BIT31 := FALSE;
   STATUS[185].EXT.ModeBit1 := FALSE;
   STATUS[185].EXT.ModeBit2 := FALSE;
   STATUS[185].EXT.ModeBit3 := FALSE;
   STATUS[185].EXT.BIT19 := FALSE;
   STATUS[185].EXT.BIT20 := FALSE;
   STATUS[185].EXT.AlarmSuppressed := FALSE;
   STATUS[185].EXT.AlarmPresent := FALSE;
   STATUS[185].EXT.AlarmFailUnAck := FALSE;
   STATUS[185].Status := 0;
   STATUS[185].TimeStamp := 16#0000;
   STATUS[186].EXT.AlarmWarnUnAck := FALSE;
   STATUS[186].EXT.AckRequired := FALSE;
   STATUS[186].EXT.Maintanence := FALSE;
   STATUS[186].EXT.Operation := FALSE;
   STATUS[186].EXT.Forced := FALSE;
   STATUS[186].EXT.BIT29 := FALSE;
   STATUS[186].EXT.BIT30 := FALSE;
   STATUS[186].EXT.BIT31 := FALSE;
   STATUS[186].EXT.ModeBit1 := FALSE;
   STATUS[186].EXT.ModeBit2 := FALSE;
   STATUS[186].EXT.ModeBit3 := FALSE;
   STATUS[186].EXT.BIT19 := FALSE;
   STATUS[186].EXT.BIT20 := FALSE;
   STATUS[186].EXT.AlarmSuppressed := FALSE;
   STATUS[186].EXT.AlarmPresent := FALSE;
   STATUS[186].EXT.AlarmFailUnAck := FALSE;
   STATUS[186].Status := 0;
   STATUS[186].TimeStamp := 16#0000;
   STATUS[187].EXT.AlarmWarnUnAck := FALSE;
   STATUS[187].EXT.AckRequired := FALSE;
   STATUS[187].EXT.Maintanence := FALSE;
   STATUS[187].EXT.Operation := FALSE;
   STATUS[187].EXT.Forced := FALSE;
   STATUS[187].EXT.BIT29 := FALSE;
   STATUS[187].EXT.BIT30 := FALSE;
   STATUS[187].EXT.BIT31 := FALSE;
   STATUS[187].EXT.ModeBit1 := FALSE;
   STATUS[187].EXT.ModeBit2 := FALSE;
   STATUS[187].EXT.ModeBit3 := FALSE;
   STATUS[187].EXT.BIT19 := FALSE;
   STATUS[187].EXT.BIT20 := FALSE;
   STATUS[187].EXT.AlarmSuppressed := FALSE;
   STATUS[187].EXT.AlarmPresent := FALSE;
   STATUS[187].EXT.AlarmFailUnAck := FALSE;
   STATUS[187].Status := 0;
   STATUS[187].TimeStamp := 16#0000;
   STATUS[188].EXT.AlarmWarnUnAck := FALSE;
   STATUS[188].EXT.AckRequired := FALSE;
   STATUS[188].EXT.Maintanence := FALSE;
   STATUS[188].EXT.Operation := FALSE;
   STATUS[188].EXT.Forced := FALSE;
   STATUS[188].EXT.BIT29 := FALSE;
   STATUS[188].EXT.BIT30 := FALSE;
   STATUS[188].EXT.BIT31 := FALSE;
   STATUS[188].EXT.ModeBit1 := FALSE;
   STATUS[188].EXT.ModeBit2 := FALSE;
   STATUS[188].EXT.ModeBit3 := FALSE;
   STATUS[188].EXT.BIT19 := FALSE;
   STATUS[188].EXT.BIT20 := FALSE;
   STATUS[188].EXT.AlarmSuppressed := FALSE;
   STATUS[188].EXT.AlarmPresent := FALSE;
   STATUS[188].EXT.AlarmFailUnAck := FALSE;
   STATUS[188].Status := 0;
   STATUS[188].TimeStamp := 16#0000;
   STATUS[189].EXT.AlarmWarnUnAck := FALSE;
   STATUS[189].EXT.AckRequired := FALSE;
   STATUS[189].EXT.Maintanence := FALSE;
   STATUS[189].EXT.Operation := FALSE;
   STATUS[189].EXT.Forced := FALSE;
   STATUS[189].EXT.BIT29 := FALSE;
   STATUS[189].EXT.BIT30 := FALSE;
   STATUS[189].EXT.BIT31 := FALSE;
   STATUS[189].EXT.ModeBit1 := FALSE;
   STATUS[189].EXT.ModeBit2 := FALSE;
   STATUS[189].EXT.ModeBit3 := FALSE;
   STATUS[189].EXT.BIT19 := FALSE;
   STATUS[189].EXT.BIT20 := FALSE;
   STATUS[189].EXT.AlarmSuppressed := FALSE;
   STATUS[189].EXT.AlarmPresent := FALSE;
   STATUS[189].EXT.AlarmFailUnAck := FALSE;
   STATUS[189].Status := 0;
   STATUS[189].TimeStamp := 16#0000;
   STATUS[190].EXT.AlarmWarnUnAck := FALSE;
   STATUS[190].EXT.AckRequired := FALSE;
   STATUS[190].EXT.Maintanence := FALSE;
   STATUS[190].EXT.Operation := FALSE;
   STATUS[190].EXT.Forced := FALSE;
   STATUS[190].EXT.BIT29 := FALSE;
   STATUS[190].EXT.BIT30 := FALSE;
   STATUS[190].EXT.BIT31 := FALSE;
   STATUS[190].EXT.ModeBit1 := FALSE;
   STATUS[190].EXT.ModeBit2 := FALSE;
   STATUS[190].EXT.ModeBit3 := FALSE;
   STATUS[190].EXT.BIT19 := FALSE;
   STATUS[190].EXT.BIT20 := FALSE;
   STATUS[190].EXT.AlarmSuppressed := FALSE;
   STATUS[190].EXT.AlarmPresent := FALSE;
   STATUS[190].EXT.AlarmFailUnAck := FALSE;
   STATUS[190].Status := 0;
   STATUS[190].TimeStamp := 16#0000;
   STATUS[191].EXT.AlarmWarnUnAck := FALSE;
   STATUS[191].EXT.AckRequired := FALSE;
   STATUS[191].EXT.Maintanence := FALSE;
   STATUS[191].EXT.Operation := FALSE;
   STATUS[191].EXT.Forced := FALSE;
   STATUS[191].EXT.BIT29 := FALSE;
   STATUS[191].EXT.BIT30 := FALSE;
   STATUS[191].EXT.BIT31 := FALSE;
   STATUS[191].EXT.ModeBit1 := FALSE;
   STATUS[191].EXT.ModeBit2 := FALSE;
   STATUS[191].EXT.ModeBit3 := FALSE;
   STATUS[191].EXT.BIT19 := FALSE;
   STATUS[191].EXT.BIT20 := FALSE;
   STATUS[191].EXT.AlarmSuppressed := FALSE;
   STATUS[191].EXT.AlarmPresent := FALSE;
   STATUS[191].EXT.AlarmFailUnAck := FALSE;
   STATUS[191].Status := 0;
   STATUS[191].TimeStamp := 16#0000;
   STATUS[192].EXT.AlarmWarnUnAck := FALSE;
   STATUS[192].EXT.AckRequired := FALSE;
   STATUS[192].EXT.Maintanence := FALSE;
   STATUS[192].EXT.Operation := FALSE;
   STATUS[192].EXT.Forced := FALSE;
   STATUS[192].EXT.BIT29 := FALSE;
   STATUS[192].EXT.BIT30 := FALSE;
   STATUS[192].EXT.BIT31 := FALSE;
   STATUS[192].EXT.ModeBit1 := FALSE;
   STATUS[192].EXT.ModeBit2 := FALSE;
   STATUS[192].EXT.ModeBit3 := FALSE;
   STATUS[192].EXT.BIT19 := FALSE;
   STATUS[192].EXT.BIT20 := FALSE;
   STATUS[192].EXT.AlarmSuppressed := FALSE;
   STATUS[192].EXT.AlarmPresent := FALSE;
   STATUS[192].EXT.AlarmFailUnAck := FALSE;
   STATUS[192].Status := 0;
   STATUS[192].TimeStamp := 16#0000;
   STATUS[193].EXT.AlarmWarnUnAck := FALSE;
   STATUS[193].EXT.AckRequired := FALSE;
   STATUS[193].EXT.Maintanence := FALSE;
   STATUS[193].EXT.Operation := FALSE;
   STATUS[193].EXT.Forced := FALSE;
   STATUS[193].EXT.BIT29 := FALSE;
   STATUS[193].EXT.BIT30 := FALSE;
   STATUS[193].EXT.BIT31 := FALSE;
   STATUS[193].EXT.ModeBit1 := FALSE;
   STATUS[193].EXT.ModeBit2 := FALSE;
   STATUS[193].EXT.ModeBit3 := FALSE;
   STATUS[193].EXT.BIT19 := FALSE;
   STATUS[193].EXT.BIT20 := FALSE;
   STATUS[193].EXT.AlarmSuppressed := FALSE;
   STATUS[193].EXT.AlarmPresent := FALSE;
   STATUS[193].EXT.AlarmFailUnAck := FALSE;
   STATUS[193].Status := 0;
   STATUS[193].TimeStamp := 16#0000;
   STATUS[194].EXT.AlarmWarnUnAck := FALSE;
   STATUS[194].EXT.AckRequired := FALSE;
   STATUS[194].EXT.Maintanence := FALSE;
   STATUS[194].EXT.Operation := FALSE;
   STATUS[194].EXT.Forced := FALSE;
   STATUS[194].EXT.BIT29 := FALSE;
   STATUS[194].EXT.BIT30 := FALSE;
   STATUS[194].EXT.BIT31 := FALSE;
   STATUS[194].EXT.ModeBit1 := FALSE;
   STATUS[194].EXT.ModeBit2 := FALSE;
   STATUS[194].EXT.ModeBit3 := FALSE;
   STATUS[194].EXT.BIT19 := FALSE;
   STATUS[194].EXT.BIT20 := FALSE;
   STATUS[194].EXT.AlarmSuppressed := FALSE;
   STATUS[194].EXT.AlarmPresent := FALSE;
   STATUS[194].EXT.AlarmFailUnAck := FALSE;
   STATUS[194].Status := 0;
   STATUS[194].TimeStamp := 16#0000;
   STATUS[195].EXT.AlarmWarnUnAck := FALSE;
   STATUS[195].EXT.AckRequired := FALSE;
   STATUS[195].EXT.Maintanence := FALSE;
   STATUS[195].EXT.Operation := FALSE;
   STATUS[195].EXT.Forced := FALSE;
   STATUS[195].EXT.BIT29 := FALSE;
   STATUS[195].EXT.BIT30 := FALSE;
   STATUS[195].EXT.BIT31 := FALSE;
   STATUS[195].EXT.ModeBit1 := FALSE;
   STATUS[195].EXT.ModeBit2 := FALSE;
   STATUS[195].EXT.ModeBit3 := FALSE;
   STATUS[195].EXT.BIT19 := FALSE;
   STATUS[195].EXT.BIT20 := FALSE;
   STATUS[195].EXT.AlarmSuppressed := FALSE;
   STATUS[195].EXT.AlarmPresent := FALSE;
   STATUS[195].EXT.AlarmFailUnAck := FALSE;
   STATUS[195].Status := 0;
   STATUS[195].TimeStamp := 16#0000;
   STATUS[196].EXT.AlarmWarnUnAck := FALSE;
   STATUS[196].EXT.AckRequired := FALSE;
   STATUS[196].EXT.Maintanence := FALSE;
   STATUS[196].EXT.Operation := FALSE;
   STATUS[196].EXT.Forced := FALSE;
   STATUS[196].EXT.BIT29 := FALSE;
   STATUS[196].EXT.BIT30 := FALSE;
   STATUS[196].EXT.BIT31 := FALSE;
   STATUS[196].EXT.ModeBit1 := FALSE;
   STATUS[196].EXT.ModeBit2 := FALSE;
   STATUS[196].EXT.ModeBit3 := FALSE;
   STATUS[196].EXT.BIT19 := FALSE;
   STATUS[196].EXT.BIT20 := FALSE;
   STATUS[196].EXT.AlarmSuppressed := FALSE;
   STATUS[196].EXT.AlarmPresent := FALSE;
   STATUS[196].EXT.AlarmFailUnAck := FALSE;
   STATUS[196].Status := 0;
   STATUS[196].TimeStamp := 16#0000;
   STATUS[197].EXT.AlarmWarnUnAck := FALSE;
   STATUS[197].EXT.AckRequired := FALSE;
   STATUS[197].EXT.Maintanence := FALSE;
   STATUS[197].EXT.Operation := FALSE;
   STATUS[197].EXT.Forced := FALSE;
   STATUS[197].EXT.BIT29 := FALSE;
   STATUS[197].EXT.BIT30 := FALSE;
   STATUS[197].EXT.BIT31 := FALSE;
   STATUS[197].EXT.ModeBit1 := FALSE;
   STATUS[197].EXT.ModeBit2 := FALSE;
   STATUS[197].EXT.ModeBit3 := FALSE;
   STATUS[197].EXT.BIT19 := FALSE;
   STATUS[197].EXT.BIT20 := FALSE;
   STATUS[197].EXT.AlarmSuppressed := FALSE;
   STATUS[197].EXT.AlarmPresent := FALSE;
   STATUS[197].EXT.AlarmFailUnAck := FALSE;
   STATUS[197].Status := 0;
   STATUS[197].TimeStamp := 16#0000;
   STATUS[198].EXT.AlarmWarnUnAck := FALSE;
   STATUS[198].EXT.AckRequired := FALSE;
   STATUS[198].EXT.Maintanence := FALSE;
   STATUS[198].EXT.Operation := FALSE;
   STATUS[198].EXT.Forced := FALSE;
   STATUS[198].EXT.BIT29 := FALSE;
   STATUS[198].EXT.BIT30 := FALSE;
   STATUS[198].EXT.BIT31 := FALSE;
   STATUS[198].EXT.ModeBit1 := FALSE;
   STATUS[198].EXT.ModeBit2 := FALSE;
   STATUS[198].EXT.ModeBit3 := FALSE;
   STATUS[198].EXT.BIT19 := FALSE;
   STATUS[198].EXT.BIT20 := FALSE;
   STATUS[198].EXT.AlarmSuppressed := FALSE;
   STATUS[198].EXT.AlarmPresent := FALSE;
   STATUS[198].EXT.AlarmFailUnAck := FALSE;
   STATUS[198].Status := 0;
   STATUS[198].TimeStamp := 16#0000;
   STATUS[199].EXT.AlarmWarnUnAck := FALSE;
   STATUS[199].EXT.AckRequired := FALSE;
   STATUS[199].EXT.Maintanence := FALSE;
   STATUS[199].EXT.Operation := FALSE;
   STATUS[199].EXT.Forced := FALSE;
   STATUS[199].EXT.BIT29 := FALSE;
   STATUS[199].EXT.BIT30 := FALSE;
   STATUS[199].EXT.BIT31 := FALSE;
   STATUS[199].EXT.ModeBit1 := FALSE;
   STATUS[199].EXT.ModeBit2 := FALSE;
   STATUS[199].EXT.ModeBit3 := FALSE;
   STATUS[199].EXT.BIT19 := FALSE;
   STATUS[199].EXT.BIT20 := FALSE;
   STATUS[199].EXT.AlarmSuppressed := FALSE;
   STATUS[199].EXT.AlarmPresent := FALSE;
   STATUS[199].EXT.AlarmFailUnAck := FALSE;
   STATUS[199].Status := 0;
   STATUS[199].TimeStamp := 16#0000;
   STATUS[200].EXT.AlarmWarnUnAck := FALSE;
   STATUS[200].EXT.AckRequired := FALSE;
   STATUS[200].EXT.Maintanence := FALSE;
   STATUS[200].EXT.Operation := FALSE;
   STATUS[200].EXT.Forced := FALSE;
   STATUS[200].EXT.BIT29 := FALSE;
   STATUS[200].EXT.BIT30 := FALSE;
   STATUS[200].EXT.BIT31 := FALSE;
   STATUS[200].EXT.ModeBit1 := FALSE;
   STATUS[200].EXT.ModeBit2 := FALSE;
   STATUS[200].EXT.ModeBit3 := FALSE;
   STATUS[200].EXT.BIT19 := FALSE;
   STATUS[200].EXT.BIT20 := FALSE;
   STATUS[200].EXT.AlarmSuppressed := FALSE;
   STATUS[200].EXT.AlarmPresent := FALSE;
   STATUS[200].EXT.AlarmFailUnAck := FALSE;
   STATUS[200].Status := 0;
   STATUS[200].TimeStamp := 16#0000;
   STATUS[201].EXT.AlarmWarnUnAck := FALSE;
   STATUS[201].EXT.AckRequired := FALSE;
   STATUS[201].EXT.Maintanence := FALSE;
   STATUS[201].EXT.Operation := FALSE;
   STATUS[201].EXT.Forced := FALSE;
   STATUS[201].EXT.BIT29 := FALSE;
   STATUS[201].EXT.BIT30 := FALSE;
   STATUS[201].EXT.BIT31 := FALSE;
   STATUS[201].EXT.ModeBit1 := FALSE;
   STATUS[201].EXT.ModeBit2 := FALSE;
   STATUS[201].EXT.ModeBit3 := FALSE;
   STATUS[201].EXT.BIT19 := FALSE;
   STATUS[201].EXT.BIT20 := FALSE;
   STATUS[201].EXT.AlarmSuppressed := FALSE;
   STATUS[201].EXT.AlarmPresent := FALSE;
   STATUS[201].EXT.AlarmFailUnAck := FALSE;
   STATUS[201].Status := 0;
   STATUS[201].TimeStamp := 16#0000;
   STATUS[202].EXT.AlarmWarnUnAck := FALSE;
   STATUS[202].EXT.AckRequired := FALSE;
   STATUS[202].EXT.Maintanence := FALSE;
   STATUS[202].EXT.Operation := FALSE;
   STATUS[202].EXT.Forced := FALSE;
   STATUS[202].EXT.BIT29 := FALSE;
   STATUS[202].EXT.BIT30 := FALSE;
   STATUS[202].EXT.BIT31 := FALSE;
   STATUS[202].EXT.ModeBit1 := FALSE;
   STATUS[202].EXT.ModeBit2 := FALSE;
   STATUS[202].EXT.ModeBit3 := FALSE;
   STATUS[202].EXT.BIT19 := FALSE;
   STATUS[202].EXT.BIT20 := FALSE;
   STATUS[202].EXT.AlarmSuppressed := FALSE;
   STATUS[202].EXT.AlarmPresent := FALSE;
   STATUS[202].EXT.AlarmFailUnAck := FALSE;
   STATUS[202].Status := 0;
   STATUS[202].TimeStamp := 16#0000;
   STATUS[203].EXT.AlarmWarnUnAck := FALSE;
   STATUS[203].EXT.AckRequired := FALSE;
   STATUS[203].EXT.Maintanence := FALSE;
   STATUS[203].EXT.Operation := FALSE;
   STATUS[203].EXT.Forced := FALSE;
   STATUS[203].EXT.BIT29 := FALSE;
   STATUS[203].EXT.BIT30 := FALSE;
   STATUS[203].EXT.BIT31 := FALSE;
   STATUS[203].EXT.ModeBit1 := FALSE;
   STATUS[203].EXT.ModeBit2 := FALSE;
   STATUS[203].EXT.ModeBit3 := FALSE;
   STATUS[203].EXT.BIT19 := FALSE;
   STATUS[203].EXT.BIT20 := FALSE;
   STATUS[203].EXT.AlarmSuppressed := FALSE;
   STATUS[203].EXT.AlarmPresent := FALSE;
   STATUS[203].EXT.AlarmFailUnAck := FALSE;
   STATUS[203].Status := 0;
   STATUS[203].TimeStamp := 16#0000;
   STATUS[204].EXT.AlarmWarnUnAck := FALSE;
   STATUS[204].EXT.AckRequired := FALSE;
   STATUS[204].EXT.Maintanence := FALSE;
   STATUS[204].EXT.Operation := FALSE;
   STATUS[204].EXT.Forced := FALSE;
   STATUS[204].EXT.BIT29 := FALSE;
   STATUS[204].EXT.BIT30 := FALSE;
   STATUS[204].EXT.BIT31 := FALSE;
   STATUS[204].EXT.ModeBit1 := FALSE;
   STATUS[204].EXT.ModeBit2 := FALSE;
   STATUS[204].EXT.ModeBit3 := FALSE;
   STATUS[204].EXT.BIT19 := FALSE;
   STATUS[204].EXT.BIT20 := FALSE;
   STATUS[204].EXT.AlarmSuppressed := FALSE;
   STATUS[204].EXT.AlarmPresent := FALSE;
   STATUS[204].EXT.AlarmFailUnAck := FALSE;
   STATUS[204].Status := 0;
   STATUS[204].TimeStamp := 16#0000;
   STATUS[205].EXT.AlarmWarnUnAck := FALSE;
   STATUS[205].EXT.AckRequired := FALSE;
   STATUS[205].EXT.Maintanence := FALSE;
   STATUS[205].EXT.Operation := FALSE;
   STATUS[205].EXT.Forced := FALSE;
   STATUS[205].EXT.BIT29 := FALSE;
   STATUS[205].EXT.BIT30 := FALSE;
   STATUS[205].EXT.BIT31 := FALSE;
   STATUS[205].EXT.ModeBit1 := FALSE;
   STATUS[205].EXT.ModeBit2 := FALSE;
   STATUS[205].EXT.ModeBit3 := FALSE;
   STATUS[205].EXT.BIT19 := FALSE;
   STATUS[205].EXT.BIT20 := FALSE;
   STATUS[205].EXT.AlarmSuppressed := FALSE;
   STATUS[205].EXT.AlarmPresent := FALSE;
   STATUS[205].EXT.AlarmFailUnAck := FALSE;
   STATUS[205].Status := 0;
   STATUS[205].TimeStamp := 16#0000;
   STATUS[206].EXT.AlarmWarnUnAck := FALSE;
   STATUS[206].EXT.AckRequired := FALSE;
   STATUS[206].EXT.Maintanence := FALSE;
   STATUS[206].EXT.Operation := FALSE;
   STATUS[206].EXT.Forced := FALSE;
   STATUS[206].EXT.BIT29 := FALSE;
   STATUS[206].EXT.BIT30 := FALSE;
   STATUS[206].EXT.BIT31 := FALSE;
   STATUS[206].EXT.ModeBit1 := FALSE;
   STATUS[206].EXT.ModeBit2 := FALSE;
   STATUS[206].EXT.ModeBit3 := FALSE;
   STATUS[206].EXT.BIT19 := FALSE;
   STATUS[206].EXT.BIT20 := FALSE;
   STATUS[206].EXT.AlarmSuppressed := FALSE;
   STATUS[206].EXT.AlarmPresent := FALSE;
   STATUS[206].EXT.AlarmFailUnAck := FALSE;
   STATUS[206].Status := 0;
   STATUS[206].TimeStamp := 16#0000;
   STATUS[207].EXT.AlarmWarnUnAck := FALSE;
   STATUS[207].EXT.AckRequired := FALSE;
   STATUS[207].EXT.Maintanence := FALSE;
   STATUS[207].EXT.Operation := FALSE;
   STATUS[207].EXT.Forced := FALSE;
   STATUS[207].EXT.BIT29 := FALSE;
   STATUS[207].EXT.BIT30 := FALSE;
   STATUS[207].EXT.BIT31 := FALSE;
   STATUS[207].EXT.ModeBit1 := FALSE;
   STATUS[207].EXT.ModeBit2 := FALSE;
   STATUS[207].EXT.ModeBit3 := FALSE;
   STATUS[207].EXT.BIT19 := FALSE;
   STATUS[207].EXT.BIT20 := FALSE;
   STATUS[207].EXT.AlarmSuppressed := FALSE;
   STATUS[207].EXT.AlarmPresent := FALSE;
   STATUS[207].EXT.AlarmFailUnAck := FALSE;
   STATUS[207].Status := 0;
   STATUS[207].TimeStamp := 16#0000;
   STATUS[208].EXT.AlarmWarnUnAck := FALSE;
   STATUS[208].EXT.AckRequired := FALSE;
   STATUS[208].EXT.Maintanence := FALSE;
   STATUS[208].EXT.Operation := FALSE;
   STATUS[208].EXT.Forced := FALSE;
   STATUS[208].EXT.BIT29 := FALSE;
   STATUS[208].EXT.BIT30 := FALSE;
   STATUS[208].EXT.BIT31 := FALSE;
   STATUS[208].EXT.ModeBit1 := FALSE;
   STATUS[208].EXT.ModeBit2 := FALSE;
   STATUS[208].EXT.ModeBit3 := FALSE;
   STATUS[208].EXT.BIT19 := FALSE;
   STATUS[208].EXT.BIT20 := FALSE;
   STATUS[208].EXT.AlarmSuppressed := FALSE;
   STATUS[208].EXT.AlarmPresent := FALSE;
   STATUS[208].EXT.AlarmFailUnAck := FALSE;
   STATUS[208].Status := 0;
   STATUS[208].TimeStamp := 16#0000;
   STATUS[209].EXT.AlarmWarnUnAck := FALSE;
   STATUS[209].EXT.AckRequired := FALSE;
   STATUS[209].EXT.Maintanence := FALSE;
   STATUS[209].EXT.Operation := FALSE;
   STATUS[209].EXT.Forced := FALSE;
   STATUS[209].EXT.BIT29 := FALSE;
   STATUS[209].EXT.BIT30 := FALSE;
   STATUS[209].EXT.BIT31 := FALSE;
   STATUS[209].EXT.ModeBit1 := FALSE;
   STATUS[209].EXT.ModeBit2 := FALSE;
   STATUS[209].EXT.ModeBit3 := FALSE;
   STATUS[209].EXT.BIT19 := FALSE;
   STATUS[209].EXT.BIT20 := FALSE;
   STATUS[209].EXT.AlarmSuppressed := FALSE;
   STATUS[209].EXT.AlarmPresent := FALSE;
   STATUS[209].EXT.AlarmFailUnAck := FALSE;
   STATUS[209].Status := 0;
   STATUS[209].TimeStamp := 16#0000;
   STATUS[210].EXT.AlarmWarnUnAck := FALSE;
   STATUS[210].EXT.AckRequired := FALSE;
   STATUS[210].EXT.Maintanence := FALSE;
   STATUS[210].EXT.Operation := FALSE;
   STATUS[210].EXT.Forced := FALSE;
   STATUS[210].EXT.BIT29 := FALSE;
   STATUS[210].EXT.BIT30 := FALSE;
   STATUS[210].EXT.BIT31 := FALSE;
   STATUS[210].EXT.ModeBit1 := FALSE;
   STATUS[210].EXT.ModeBit2 := FALSE;
   STATUS[210].EXT.ModeBit3 := FALSE;
   STATUS[210].EXT.BIT19 := FALSE;
   STATUS[210].EXT.BIT20 := FALSE;
   STATUS[210].EXT.AlarmSuppressed := FALSE;
   STATUS[210].EXT.AlarmPresent := FALSE;
   STATUS[210].EXT.AlarmFailUnAck := FALSE;
   STATUS[210].Status := 0;
   STATUS[210].TimeStamp := 16#0000;
   STATUS[211].EXT.AlarmWarnUnAck := FALSE;
   STATUS[211].EXT.AckRequired := FALSE;
   STATUS[211].EXT.Maintanence := FALSE;
   STATUS[211].EXT.Operation := FALSE;
   STATUS[211].EXT.Forced := FALSE;
   STATUS[211].EXT.BIT29 := FALSE;
   STATUS[211].EXT.BIT30 := FALSE;
   STATUS[211].EXT.BIT31 := FALSE;
   STATUS[211].EXT.ModeBit1 := FALSE;
   STATUS[211].EXT.ModeBit2 := FALSE;
   STATUS[211].EXT.ModeBit3 := FALSE;
   STATUS[211].EXT.BIT19 := FALSE;
   STATUS[211].EXT.BIT20 := FALSE;
   STATUS[211].EXT.AlarmSuppressed := FALSE;
   STATUS[211].EXT.AlarmPresent := FALSE;
   STATUS[211].EXT.AlarmFailUnAck := FALSE;
   STATUS[211].Status := 0;
   STATUS[211].TimeStamp := 16#0000;
   STATUS[212].EXT.AlarmWarnUnAck := FALSE;
   STATUS[212].EXT.AckRequired := FALSE;
   STATUS[212].EXT.Maintanence := FALSE;
   STATUS[212].EXT.Operation := FALSE;
   STATUS[212].EXT.Forced := FALSE;
   STATUS[212].EXT.BIT29 := FALSE;
   STATUS[212].EXT.BIT30 := FALSE;
   STATUS[212].EXT.BIT31 := FALSE;
   STATUS[212].EXT.ModeBit1 := FALSE;
   STATUS[212].EXT.ModeBit2 := FALSE;
   STATUS[212].EXT.ModeBit3 := FALSE;
   STATUS[212].EXT.BIT19 := FALSE;
   STATUS[212].EXT.BIT20 := FALSE;
   STATUS[212].EXT.AlarmSuppressed := FALSE;
   STATUS[212].EXT.AlarmPresent := FALSE;
   STATUS[212].EXT.AlarmFailUnAck := FALSE;
   STATUS[212].Status := 0;
   STATUS[212].TimeStamp := 16#0000;
   STATUS[213].EXT.AlarmWarnUnAck := FALSE;
   STATUS[213].EXT.AckRequired := FALSE;
   STATUS[213].EXT.Maintanence := FALSE;
   STATUS[213].EXT.Operation := FALSE;
   STATUS[213].EXT.Forced := FALSE;
   STATUS[213].EXT.BIT29 := FALSE;
   STATUS[213].EXT.BIT30 := FALSE;
   STATUS[213].EXT.BIT31 := FALSE;
   STATUS[213].EXT.ModeBit1 := FALSE;
   STATUS[213].EXT.ModeBit2 := FALSE;
   STATUS[213].EXT.ModeBit3 := FALSE;
   STATUS[213].EXT.BIT19 := FALSE;
   STATUS[213].EXT.BIT20 := FALSE;
   STATUS[213].EXT.AlarmSuppressed := FALSE;
   STATUS[213].EXT.AlarmPresent := FALSE;
   STATUS[213].EXT.AlarmFailUnAck := FALSE;
   STATUS[213].Status := 0;
   STATUS[213].TimeStamp := 16#0000;
   STATUS[214].EXT.AlarmWarnUnAck := FALSE;
   STATUS[214].EXT.AckRequired := FALSE;
   STATUS[214].EXT.Maintanence := FALSE;
   STATUS[214].EXT.Operation := FALSE;
   STATUS[214].EXT.Forced := FALSE;
   STATUS[214].EXT.BIT29 := FALSE;
   STATUS[214].EXT.BIT30 := FALSE;
   STATUS[214].EXT.BIT31 := FALSE;
   STATUS[214].EXT.ModeBit1 := FALSE;
   STATUS[214].EXT.ModeBit2 := FALSE;
   STATUS[214].EXT.ModeBit3 := FALSE;
   STATUS[214].EXT.BIT19 := FALSE;
   STATUS[214].EXT.BIT20 := FALSE;
   STATUS[214].EXT.AlarmSuppressed := FALSE;
   STATUS[214].EXT.AlarmPresent := FALSE;
   STATUS[214].EXT.AlarmFailUnAck := FALSE;
   STATUS[214].Status := 0;
   STATUS[214].TimeStamp := 16#0000;
   STATUS[215].EXT.AlarmWarnUnAck := FALSE;
   STATUS[215].EXT.AckRequired := FALSE;
   STATUS[215].EXT.Maintanence := FALSE;
   STATUS[215].EXT.Operation := FALSE;
   STATUS[215].EXT.Forced := FALSE;
   STATUS[215].EXT.BIT29 := FALSE;
   STATUS[215].EXT.BIT30 := FALSE;
   STATUS[215].EXT.BIT31 := FALSE;
   STATUS[215].EXT.ModeBit1 := FALSE;
   STATUS[215].EXT.ModeBit2 := FALSE;
   STATUS[215].EXT.ModeBit3 := FALSE;
   STATUS[215].EXT.BIT19 := FALSE;
   STATUS[215].EXT.BIT20 := FALSE;
   STATUS[215].EXT.AlarmSuppressed := FALSE;
   STATUS[215].EXT.AlarmPresent := FALSE;
   STATUS[215].EXT.AlarmFailUnAck := FALSE;
   STATUS[215].Status := 0;
   STATUS[215].TimeStamp := 16#0000;
   STATUS[216].EXT.AlarmWarnUnAck := FALSE;
   STATUS[216].EXT.AckRequired := FALSE;
   STATUS[216].EXT.Maintanence := FALSE;
   STATUS[216].EXT.Operation := FALSE;
   STATUS[216].EXT.Forced := FALSE;
   STATUS[216].EXT.BIT29 := FALSE;
   STATUS[216].EXT.BIT30 := FALSE;
   STATUS[216].EXT.BIT31 := FALSE;
   STATUS[216].EXT.ModeBit1 := FALSE;
   STATUS[216].EXT.ModeBit2 := FALSE;
   STATUS[216].EXT.ModeBit3 := FALSE;
   STATUS[216].EXT.BIT19 := FALSE;
   STATUS[216].EXT.BIT20 := FALSE;
   STATUS[216].EXT.AlarmSuppressed := FALSE;
   STATUS[216].EXT.AlarmPresent := FALSE;
   STATUS[216].EXT.AlarmFailUnAck := FALSE;
   STATUS[216].Status := 0;
   STATUS[216].TimeStamp := 16#0000;
   STATUS[217].EXT.AlarmWarnUnAck := FALSE;
   STATUS[217].EXT.AckRequired := FALSE;
   STATUS[217].EXT.Maintanence := FALSE;
   STATUS[217].EXT.Operation := FALSE;
   STATUS[217].EXT.Forced := FALSE;
   STATUS[217].EXT.BIT29 := FALSE;
   STATUS[217].EXT.BIT30 := FALSE;
   STATUS[217].EXT.BIT31 := FALSE;
   STATUS[217].EXT.ModeBit1 := FALSE;
   STATUS[217].EXT.ModeBit2 := FALSE;
   STATUS[217].EXT.ModeBit3 := FALSE;
   STATUS[217].EXT.BIT19 := FALSE;
   STATUS[217].EXT.BIT20 := FALSE;
   STATUS[217].EXT.AlarmSuppressed := FALSE;
   STATUS[217].EXT.AlarmPresent := FALSE;
   STATUS[217].EXT.AlarmFailUnAck := FALSE;
   STATUS[217].Status := 0;
   STATUS[217].TimeStamp := 16#0000;
   STATUS[218].EXT.AlarmWarnUnAck := FALSE;
   STATUS[218].EXT.AckRequired := FALSE;
   STATUS[218].EXT.Maintanence := FALSE;
   STATUS[218].EXT.Operation := FALSE;
   STATUS[218].EXT.Forced := FALSE;
   STATUS[218].EXT.BIT29 := FALSE;
   STATUS[218].EXT.BIT30 := FALSE;
   STATUS[218].EXT.BIT31 := FALSE;
   STATUS[218].EXT.ModeBit1 := FALSE;
   STATUS[218].EXT.ModeBit2 := FALSE;
   STATUS[218].EXT.ModeBit3 := FALSE;
   STATUS[218].EXT.BIT19 := FALSE;
   STATUS[218].EXT.BIT20 := FALSE;
   STATUS[218].EXT.AlarmSuppressed := FALSE;
   STATUS[218].EXT.AlarmPresent := FALSE;
   STATUS[218].EXT.AlarmFailUnAck := FALSE;
   STATUS[218].Status := 0;
   STATUS[218].TimeStamp := 16#0000;
   STATUS[219].EXT.AlarmWarnUnAck := FALSE;
   STATUS[219].EXT.AckRequired := FALSE;
   STATUS[219].EXT.Maintanence := FALSE;
   STATUS[219].EXT.Operation := FALSE;
   STATUS[219].EXT.Forced := FALSE;
   STATUS[219].EXT.BIT29 := FALSE;
   STATUS[219].EXT.BIT30 := FALSE;
   STATUS[219].EXT.BIT31 := FALSE;
   STATUS[219].EXT.ModeBit1 := FALSE;
   STATUS[219].EXT.ModeBit2 := FALSE;
   STATUS[219].EXT.ModeBit3 := FALSE;
   STATUS[219].EXT.BIT19 := FALSE;
   STATUS[219].EXT.BIT20 := FALSE;
   STATUS[219].EXT.AlarmSuppressed := FALSE;
   STATUS[219].EXT.AlarmPresent := FALSE;
   STATUS[219].EXT.AlarmFailUnAck := FALSE;
   STATUS[219].Status := 0;
   STATUS[219].TimeStamp := 16#0000;
   STATUS[220].EXT.AlarmWarnUnAck := FALSE;
   STATUS[220].EXT.AckRequired := FALSE;
   STATUS[220].EXT.Maintanence := FALSE;
   STATUS[220].EXT.Operation := FALSE;
   STATUS[220].EXT.Forced := FALSE;
   STATUS[220].EXT.BIT29 := FALSE;
   STATUS[220].EXT.BIT30 := FALSE;
   STATUS[220].EXT.BIT31 := FALSE;
   STATUS[220].EXT.ModeBit1 := FALSE;
   STATUS[220].EXT.ModeBit2 := FALSE;
   STATUS[220].EXT.ModeBit3 := FALSE;
   STATUS[220].EXT.BIT19 := FALSE;
   STATUS[220].EXT.BIT20 := FALSE;
   STATUS[220].EXT.AlarmSuppressed := FALSE;
   STATUS[220].EXT.AlarmPresent := FALSE;
   STATUS[220].EXT.AlarmFailUnAck := FALSE;
   STATUS[220].Status := 0;
   STATUS[220].TimeStamp := 16#0000;
   STATUS[221].EXT.AlarmWarnUnAck := FALSE;
   STATUS[221].EXT.AckRequired := FALSE;
   STATUS[221].EXT.Maintanence := FALSE;
   STATUS[221].EXT.Operation := FALSE;
   STATUS[221].EXT.Forced := FALSE;
   STATUS[221].EXT.BIT29 := FALSE;
   STATUS[221].EXT.BIT30 := FALSE;
   STATUS[221].EXT.BIT31 := FALSE;
   STATUS[221].EXT.ModeBit1 := FALSE;
   STATUS[221].EXT.ModeBit2 := FALSE;
   STATUS[221].EXT.ModeBit3 := FALSE;
   STATUS[221].EXT.BIT19 := FALSE;
   STATUS[221].EXT.BIT20 := FALSE;
   STATUS[221].EXT.AlarmSuppressed := FALSE;
   STATUS[221].EXT.AlarmPresent := FALSE;
   STATUS[221].EXT.AlarmFailUnAck := FALSE;
   STATUS[221].Status := 0;
   STATUS[221].TimeStamp := 16#0000;
   STATUS[222].EXT.AlarmWarnUnAck := FALSE;
   STATUS[222].EXT.AckRequired := FALSE;
   STATUS[222].EXT.Maintanence := FALSE;
   STATUS[222].EXT.Operation := FALSE;
   STATUS[222].EXT.Forced := FALSE;
   STATUS[222].EXT.BIT29 := FALSE;
   STATUS[222].EXT.BIT30 := FALSE;
   STATUS[222].EXT.BIT31 := FALSE;
   STATUS[222].EXT.ModeBit1 := FALSE;
   STATUS[222].EXT.ModeBit2 := FALSE;
   STATUS[222].EXT.ModeBit3 := FALSE;
   STATUS[222].EXT.BIT19 := FALSE;
   STATUS[222].EXT.BIT20 := FALSE;
   STATUS[222].EXT.AlarmSuppressed := FALSE;
   STATUS[222].EXT.AlarmPresent := FALSE;
   STATUS[222].EXT.AlarmFailUnAck := FALSE;
   STATUS[222].Status := 0;
   STATUS[222].TimeStamp := 16#0000;
   STATUS[223].EXT.AlarmWarnUnAck := FALSE;
   STATUS[223].EXT.AckRequired := FALSE;
   STATUS[223].EXT.Maintanence := FALSE;
   STATUS[223].EXT.Operation := FALSE;
   STATUS[223].EXT.Forced := FALSE;
   STATUS[223].EXT.BIT29 := FALSE;
   STATUS[223].EXT.BIT30 := FALSE;
   STATUS[223].EXT.BIT31 := FALSE;
   STATUS[223].EXT.ModeBit1 := FALSE;
   STATUS[223].EXT.ModeBit2 := FALSE;
   STATUS[223].EXT.ModeBit3 := FALSE;
   STATUS[223].EXT.BIT19 := FALSE;
   STATUS[223].EXT.BIT20 := FALSE;
   STATUS[223].EXT.AlarmSuppressed := FALSE;
   STATUS[223].EXT.AlarmPresent := FALSE;
   STATUS[223].EXT.AlarmFailUnAck := FALSE;
   STATUS[223].Status := 0;
   STATUS[223].TimeStamp := 16#0000;
   STATUS[224].EXT.AlarmWarnUnAck := FALSE;
   STATUS[224].EXT.AckRequired := FALSE;
   STATUS[224].EXT.Maintanence := FALSE;
   STATUS[224].EXT.Operation := FALSE;
   STATUS[224].EXT.Forced := FALSE;
   STATUS[224].EXT.BIT29 := FALSE;
   STATUS[224].EXT.BIT30 := FALSE;
   STATUS[224].EXT.BIT31 := FALSE;
   STATUS[224].EXT.ModeBit1 := FALSE;
   STATUS[224].EXT.ModeBit2 := FALSE;
   STATUS[224].EXT.ModeBit3 := FALSE;
   STATUS[224].EXT.BIT19 := FALSE;
   STATUS[224].EXT.BIT20 := FALSE;
   STATUS[224].EXT.AlarmSuppressed := FALSE;
   STATUS[224].EXT.AlarmPresent := FALSE;
   STATUS[224].EXT.AlarmFailUnAck := FALSE;
   STATUS[224].Status := 0;
   STATUS[224].TimeStamp := 16#0000;
   STATUS[225].EXT.AlarmWarnUnAck := FALSE;
   STATUS[225].EXT.AckRequired := FALSE;
   STATUS[225].EXT.Maintanence := FALSE;
   STATUS[225].EXT.Operation := FALSE;
   STATUS[225].EXT.Forced := FALSE;
   STATUS[225].EXT.BIT29 := FALSE;
   STATUS[225].EXT.BIT30 := FALSE;
   STATUS[225].EXT.BIT31 := FALSE;
   STATUS[225].EXT.ModeBit1 := FALSE;
   STATUS[225].EXT.ModeBit2 := FALSE;
   STATUS[225].EXT.ModeBit3 := FALSE;
   STATUS[225].EXT.BIT19 := FALSE;
   STATUS[225].EXT.BIT20 := FALSE;
   STATUS[225].EXT.AlarmSuppressed := FALSE;
   STATUS[225].EXT.AlarmPresent := FALSE;
   STATUS[225].EXT.AlarmFailUnAck := FALSE;
   STATUS[225].Status := 0;
   STATUS[225].TimeStamp := 16#0000;
   STATUS[226].EXT.AlarmWarnUnAck := FALSE;
   STATUS[226].EXT.AckRequired := FALSE;
   STATUS[226].EXT.Maintanence := FALSE;
   STATUS[226].EXT.Operation := FALSE;
   STATUS[226].EXT.Forced := FALSE;
   STATUS[226].EXT.BIT29 := FALSE;
   STATUS[226].EXT.BIT30 := FALSE;
   STATUS[226].EXT.BIT31 := FALSE;
   STATUS[226].EXT.ModeBit1 := FALSE;
   STATUS[226].EXT.ModeBit2 := FALSE;
   STATUS[226].EXT.ModeBit3 := FALSE;
   STATUS[226].EXT.BIT19 := FALSE;
   STATUS[226].EXT.BIT20 := FALSE;
   STATUS[226].EXT.AlarmSuppressed := FALSE;
   STATUS[226].EXT.AlarmPresent := FALSE;
   STATUS[226].EXT.AlarmFailUnAck := FALSE;
   STATUS[226].Status := 0;
   STATUS[226].TimeStamp := 16#0000;
   STATUS[227].EXT.AlarmWarnUnAck := FALSE;
   STATUS[227].EXT.AckRequired := FALSE;
   STATUS[227].EXT.Maintanence := FALSE;
   STATUS[227].EXT.Operation := FALSE;
   STATUS[227].EXT.Forced := FALSE;
   STATUS[227].EXT.BIT29 := FALSE;
   STATUS[227].EXT.BIT30 := FALSE;
   STATUS[227].EXT.BIT31 := FALSE;
   STATUS[227].EXT.ModeBit1 := FALSE;
   STATUS[227].EXT.ModeBit2 := FALSE;
   STATUS[227].EXT.ModeBit3 := FALSE;
   STATUS[227].EXT.BIT19 := FALSE;
   STATUS[227].EXT.BIT20 := FALSE;
   STATUS[227].EXT.AlarmSuppressed := FALSE;
   STATUS[227].EXT.AlarmPresent := FALSE;
   STATUS[227].EXT.AlarmFailUnAck := FALSE;
   STATUS[227].Status := 0;
   STATUS[227].TimeStamp := 16#0000;
   STATUS[228].EXT.AlarmWarnUnAck := FALSE;
   STATUS[228].EXT.AckRequired := FALSE;
   STATUS[228].EXT.Maintanence := FALSE;
   STATUS[228].EXT.Operation := FALSE;
   STATUS[228].EXT.Forced := FALSE;
   STATUS[228].EXT.BIT29 := FALSE;
   STATUS[228].EXT.BIT30 := FALSE;
   STATUS[228].EXT.BIT31 := FALSE;
   STATUS[228].EXT.ModeBit1 := FALSE;
   STATUS[228].EXT.ModeBit2 := FALSE;
   STATUS[228].EXT.ModeBit3 := FALSE;
   STATUS[228].EXT.BIT19 := FALSE;
   STATUS[228].EXT.BIT20 := FALSE;
   STATUS[228].EXT.AlarmSuppressed := FALSE;
   STATUS[228].EXT.AlarmPresent := FALSE;
   STATUS[228].EXT.AlarmFailUnAck := FALSE;
   STATUS[228].Status := 0;
   STATUS[228].TimeStamp := 16#0000;
   STATUS[229].EXT.AlarmWarnUnAck := FALSE;
   STATUS[229].EXT.AckRequired := FALSE;
   STATUS[229].EXT.Maintanence := FALSE;
   STATUS[229].EXT.Operation := FALSE;
   STATUS[229].EXT.Forced := FALSE;
   STATUS[229].EXT.BIT29 := FALSE;
   STATUS[229].EXT.BIT30 := FALSE;
   STATUS[229].EXT.BIT31 := FALSE;
   STATUS[229].EXT.ModeBit1 := FALSE;
   STATUS[229].EXT.ModeBit2 := FALSE;
   STATUS[229].EXT.ModeBit3 := FALSE;
   STATUS[229].EXT.BIT19 := FALSE;
   STATUS[229].EXT.BIT20 := FALSE;
   STATUS[229].EXT.AlarmSuppressed := FALSE;
   STATUS[229].EXT.AlarmPresent := FALSE;
   STATUS[229].EXT.AlarmFailUnAck := FALSE;
   STATUS[229].Status := 0;
   STATUS[229].TimeStamp := 16#0000;
   STATUS[230].EXT.AlarmWarnUnAck := FALSE;
   STATUS[230].EXT.AckRequired := FALSE;
   STATUS[230].EXT.Maintanence := FALSE;
   STATUS[230].EXT.Operation := FALSE;
   STATUS[230].EXT.Forced := FALSE;
   STATUS[230].EXT.BIT29 := FALSE;
   STATUS[230].EXT.BIT30 := FALSE;
   STATUS[230].EXT.BIT31 := FALSE;
   STATUS[230].EXT.ModeBit1 := FALSE;
   STATUS[230].EXT.ModeBit2 := FALSE;
   STATUS[230].EXT.ModeBit3 := FALSE;
   STATUS[230].EXT.BIT19 := FALSE;
   STATUS[230].EXT.BIT20 := FALSE;
   STATUS[230].EXT.AlarmSuppressed := FALSE;
   STATUS[230].EXT.AlarmPresent := FALSE;
   STATUS[230].EXT.AlarmFailUnAck := FALSE;
   STATUS[230].Status := 0;
   STATUS[230].TimeStamp := 16#0000;
   STATUS[231].EXT.AlarmWarnUnAck := FALSE;
   STATUS[231].EXT.AckRequired := FALSE;
   STATUS[231].EXT.Maintanence := FALSE;
   STATUS[231].EXT.Operation := FALSE;
   STATUS[231].EXT.Forced := FALSE;
   STATUS[231].EXT.BIT29 := FALSE;
   STATUS[231].EXT.BIT30 := FALSE;
   STATUS[231].EXT.BIT31 := FALSE;
   STATUS[231].EXT.ModeBit1 := FALSE;
   STATUS[231].EXT.ModeBit2 := FALSE;
   STATUS[231].EXT.ModeBit3 := FALSE;
   STATUS[231].EXT.BIT19 := FALSE;
   STATUS[231].EXT.BIT20 := FALSE;
   STATUS[231].EXT.AlarmSuppressed := FALSE;
   STATUS[231].EXT.AlarmPresent := FALSE;
   STATUS[231].EXT.AlarmFailUnAck := FALSE;
   STATUS[231].Status := 0;
   STATUS[231].TimeStamp := 16#0000;
   STATUS[232].EXT.AlarmWarnUnAck := FALSE;
   STATUS[232].EXT.AckRequired := FALSE;
   STATUS[232].EXT.Maintanence := FALSE;
   STATUS[232].EXT.Operation := FALSE;
   STATUS[232].EXT.Forced := FALSE;
   STATUS[232].EXT.BIT29 := FALSE;
   STATUS[232].EXT.BIT30 := FALSE;
   STATUS[232].EXT.BIT31 := FALSE;
   STATUS[232].EXT.ModeBit1 := FALSE;
   STATUS[232].EXT.ModeBit2 := FALSE;
   STATUS[232].EXT.ModeBit3 := FALSE;
   STATUS[232].EXT.BIT19 := FALSE;
   STATUS[232].EXT.BIT20 := FALSE;
   STATUS[232].EXT.AlarmSuppressed := FALSE;
   STATUS[232].EXT.AlarmPresent := FALSE;
   STATUS[232].EXT.AlarmFailUnAck := FALSE;
   STATUS[232].Status := 0;
   STATUS[232].TimeStamp := 16#0000;
   STATUS[233].EXT.AlarmWarnUnAck := FALSE;
   STATUS[233].EXT.AckRequired := FALSE;
   STATUS[233].EXT.Maintanence := FALSE;
   STATUS[233].EXT.Operation := FALSE;
   STATUS[233].EXT.Forced := FALSE;
   STATUS[233].EXT.BIT29 := FALSE;
   STATUS[233].EXT.BIT30 := FALSE;
   STATUS[233].EXT.BIT31 := FALSE;
   STATUS[233].EXT.ModeBit1 := FALSE;
   STATUS[233].EXT.ModeBit2 := FALSE;
   STATUS[233].EXT.ModeBit3 := FALSE;
   STATUS[233].EXT.BIT19 := FALSE;
   STATUS[233].EXT.BIT20 := FALSE;
   STATUS[233].EXT.AlarmSuppressed := FALSE;
   STATUS[233].EXT.AlarmPresent := FALSE;
   STATUS[233].EXT.AlarmFailUnAck := FALSE;
   STATUS[233].Status := 0;
   STATUS[233].TimeStamp := 16#0000;
   STATUS[234].EXT.AlarmWarnUnAck := FALSE;
   STATUS[234].EXT.AckRequired := FALSE;
   STATUS[234].EXT.Maintanence := FALSE;
   STATUS[234].EXT.Operation := FALSE;
   STATUS[234].EXT.Forced := FALSE;
   STATUS[234].EXT.BIT29 := FALSE;
   STATUS[234].EXT.BIT30 := FALSE;
   STATUS[234].EXT.BIT31 := FALSE;
   STATUS[234].EXT.ModeBit1 := FALSE;
   STATUS[234].EXT.ModeBit2 := FALSE;
   STATUS[234].EXT.ModeBit3 := FALSE;
   STATUS[234].EXT.BIT19 := FALSE;
   STATUS[234].EXT.BIT20 := FALSE;
   STATUS[234].EXT.AlarmSuppressed := FALSE;
   STATUS[234].EXT.AlarmPresent := FALSE;
   STATUS[234].EXT.AlarmFailUnAck := FALSE;
   STATUS[234].Status := 0;
   STATUS[234].TimeStamp := 16#0000;
   STATUS[235].EXT.AlarmWarnUnAck := FALSE;
   STATUS[235].EXT.AckRequired := FALSE;
   STATUS[235].EXT.Maintanence := FALSE;
   STATUS[235].EXT.Operation := FALSE;
   STATUS[235].EXT.Forced := FALSE;
   STATUS[235].EXT.BIT29 := FALSE;
   STATUS[235].EXT.BIT30 := FALSE;
   STATUS[235].EXT.BIT31 := FALSE;
   STATUS[235].EXT.ModeBit1 := FALSE;
   STATUS[235].EXT.ModeBit2 := FALSE;
   STATUS[235].EXT.ModeBit3 := FALSE;
   STATUS[235].EXT.BIT19 := FALSE;
   STATUS[235].EXT.BIT20 := FALSE;
   STATUS[235].EXT.AlarmSuppressed := FALSE;
   STATUS[235].EXT.AlarmPresent := FALSE;
   STATUS[235].EXT.AlarmFailUnAck := FALSE;
   STATUS[235].Status := 0;
   STATUS[235].TimeStamp := 16#0000;
   STATUS[236].EXT.AlarmWarnUnAck := FALSE;
   STATUS[236].EXT.AckRequired := FALSE;
   STATUS[236].EXT.Maintanence := FALSE;
   STATUS[236].EXT.Operation := FALSE;
   STATUS[236].EXT.Forced := FALSE;
   STATUS[236].EXT.BIT29 := FALSE;
   STATUS[236].EXT.BIT30 := FALSE;
   STATUS[236].EXT.BIT31 := FALSE;
   STATUS[236].EXT.ModeBit1 := FALSE;
   STATUS[236].EXT.ModeBit2 := FALSE;
   STATUS[236].EXT.ModeBit3 := FALSE;
   STATUS[236].EXT.BIT19 := FALSE;
   STATUS[236].EXT.BIT20 := FALSE;
   STATUS[236].EXT.AlarmSuppressed := FALSE;
   STATUS[236].EXT.AlarmPresent := FALSE;
   STATUS[236].EXT.AlarmFailUnAck := FALSE;
   STATUS[236].Status := 0;
   STATUS[236].TimeStamp := 16#0000;
   STATUS[237].EXT.AlarmWarnUnAck := FALSE;
   STATUS[237].EXT.AckRequired := FALSE;
   STATUS[237].EXT.Maintanence := FALSE;
   STATUS[237].EXT.Operation := FALSE;
   STATUS[237].EXT.Forced := FALSE;
   STATUS[237].EXT.BIT29 := FALSE;
   STATUS[237].EXT.BIT30 := FALSE;
   STATUS[237].EXT.BIT31 := FALSE;
   STATUS[237].EXT.ModeBit1 := FALSE;
   STATUS[237].EXT.ModeBit2 := FALSE;
   STATUS[237].EXT.ModeBit3 := FALSE;
   STATUS[237].EXT.BIT19 := FALSE;
   STATUS[237].EXT.BIT20 := FALSE;
   STATUS[237].EXT.AlarmSuppressed := FALSE;
   STATUS[237].EXT.AlarmPresent := FALSE;
   STATUS[237].EXT.AlarmFailUnAck := FALSE;
   STATUS[237].Status := 0;
   STATUS[237].TimeStamp := 16#0000;
   STATUS[238].EXT.AlarmWarnUnAck := FALSE;
   STATUS[238].EXT.AckRequired := FALSE;
   STATUS[238].EXT.Maintanence := FALSE;
   STATUS[238].EXT.Operation := FALSE;
   STATUS[238].EXT.Forced := FALSE;
   STATUS[238].EXT.BIT29 := FALSE;
   STATUS[238].EXT.BIT30 := FALSE;
   STATUS[238].EXT.BIT31 := FALSE;
   STATUS[238].EXT.ModeBit1 := FALSE;
   STATUS[238].EXT.ModeBit2 := FALSE;
   STATUS[238].EXT.ModeBit3 := FALSE;
   STATUS[238].EXT.BIT19 := FALSE;
   STATUS[238].EXT.BIT20 := FALSE;
   STATUS[238].EXT.AlarmSuppressed := FALSE;
   STATUS[238].EXT.AlarmPresent := FALSE;
   STATUS[238].EXT.AlarmFailUnAck := FALSE;
   STATUS[238].Status := 0;
   STATUS[238].TimeStamp := 16#0000;
   STATUS[239].EXT.AlarmWarnUnAck := FALSE;
   STATUS[239].EXT.AckRequired := FALSE;
   STATUS[239].EXT.Maintanence := FALSE;
   STATUS[239].EXT.Operation := FALSE;
   STATUS[239].EXT.Forced := FALSE;
   STATUS[239].EXT.BIT29 := FALSE;
   STATUS[239].EXT.BIT30 := FALSE;
   STATUS[239].EXT.BIT31 := FALSE;
   STATUS[239].EXT.ModeBit1 := FALSE;
   STATUS[239].EXT.ModeBit2 := FALSE;
   STATUS[239].EXT.ModeBit3 := FALSE;
   STATUS[239].EXT.BIT19 := FALSE;
   STATUS[239].EXT.BIT20 := FALSE;
   STATUS[239].EXT.AlarmSuppressed := FALSE;
   STATUS[239].EXT.AlarmPresent := FALSE;
   STATUS[239].EXT.AlarmFailUnAck := FALSE;
   STATUS[239].Status := 0;
   STATUS[239].TimeStamp := 16#0000;
   STATUS[240].EXT.AlarmWarnUnAck := FALSE;
   STATUS[240].EXT.AckRequired := FALSE;
   STATUS[240].EXT.Maintanence := FALSE;
   STATUS[240].EXT.Operation := FALSE;
   STATUS[240].EXT.Forced := FALSE;
   STATUS[240].EXT.BIT29 := FALSE;
   STATUS[240].EXT.BIT30 := FALSE;
   STATUS[240].EXT.BIT31 := FALSE;
   STATUS[240].EXT.ModeBit1 := FALSE;
   STATUS[240].EXT.ModeBit2 := FALSE;
   STATUS[240].EXT.ModeBit3 := FALSE;
   STATUS[240].EXT.BIT19 := FALSE;
   STATUS[240].EXT.BIT20 := FALSE;
   STATUS[240].EXT.AlarmSuppressed := FALSE;
   STATUS[240].EXT.AlarmPresent := FALSE;
   STATUS[240].EXT.AlarmFailUnAck := FALSE;
   STATUS[240].Status := 0;
   STATUS[240].TimeStamp := 16#0000;
   STATUS[241].EXT.AlarmWarnUnAck := FALSE;
   STATUS[241].EXT.AckRequired := FALSE;
   STATUS[241].EXT.Maintanence := FALSE;
   STATUS[241].EXT.Operation := FALSE;
   STATUS[241].EXT.Forced := FALSE;
   STATUS[241].EXT.BIT29 := FALSE;
   STATUS[241].EXT.BIT30 := FALSE;
   STATUS[241].EXT.BIT31 := FALSE;
   STATUS[241].EXT.ModeBit1 := FALSE;
   STATUS[241].EXT.ModeBit2 := FALSE;
   STATUS[241].EXT.ModeBit3 := FALSE;
   STATUS[241].EXT.BIT19 := FALSE;
   STATUS[241].EXT.BIT20 := FALSE;
   STATUS[241].EXT.AlarmSuppressed := FALSE;
   STATUS[241].EXT.AlarmPresent := FALSE;
   STATUS[241].EXT.AlarmFailUnAck := FALSE;
   STATUS[241].Status := 0;
   STATUS[241].TimeStamp := 16#0000;
   STATUS[242].EXT.AlarmWarnUnAck := FALSE;
   STATUS[242].EXT.AckRequired := FALSE;
   STATUS[242].EXT.Maintanence := FALSE;
   STATUS[242].EXT.Operation := FALSE;
   STATUS[242].EXT.Forced := FALSE;
   STATUS[242].EXT.BIT29 := FALSE;
   STATUS[242].EXT.BIT30 := FALSE;
   STATUS[242].EXT.BIT31 := FALSE;
   STATUS[242].EXT.ModeBit1 := FALSE;
   STATUS[242].EXT.ModeBit2 := FALSE;
   STATUS[242].EXT.ModeBit3 := FALSE;
   STATUS[242].EXT.BIT19 := FALSE;
   STATUS[242].EXT.BIT20 := FALSE;
   STATUS[242].EXT.AlarmSuppressed := FALSE;
   STATUS[242].EXT.AlarmPresent := FALSE;
   STATUS[242].EXT.AlarmFailUnAck := FALSE;
   STATUS[242].Status := 0;
   STATUS[242].TimeStamp := 16#0000;
   STATUS[243].EXT.AlarmWarnUnAck := FALSE;
   STATUS[243].EXT.AckRequired := FALSE;
   STATUS[243].EXT.Maintanence := FALSE;
   STATUS[243].EXT.Operation := FALSE;
   STATUS[243].EXT.Forced := FALSE;
   STATUS[243].EXT.BIT29 := FALSE;
   STATUS[243].EXT.BIT30 := FALSE;
   STATUS[243].EXT.BIT31 := FALSE;
   STATUS[243].EXT.ModeBit1 := FALSE;
   STATUS[243].EXT.ModeBit2 := FALSE;
   STATUS[243].EXT.ModeBit3 := FALSE;
   STATUS[243].EXT.BIT19 := FALSE;
   STATUS[243].EXT.BIT20 := FALSE;
   STATUS[243].EXT.AlarmSuppressed := FALSE;
   STATUS[243].EXT.AlarmPresent := FALSE;
   STATUS[243].EXT.AlarmFailUnAck := FALSE;
   STATUS[243].Status := 0;
   STATUS[243].TimeStamp := 16#0000;
   STATUS[244].EXT.AlarmWarnUnAck := FALSE;
   STATUS[244].EXT.AckRequired := FALSE;
   STATUS[244].EXT.Maintanence := FALSE;
   STATUS[244].EXT.Operation := FALSE;
   STATUS[244].EXT.Forced := FALSE;
   STATUS[244].EXT.BIT29 := FALSE;
   STATUS[244].EXT.BIT30 := FALSE;
   STATUS[244].EXT.BIT31 := FALSE;
   STATUS[244].EXT.ModeBit1 := FALSE;
   STATUS[244].EXT.ModeBit2 := FALSE;
   STATUS[244].EXT.ModeBit3 := FALSE;
   STATUS[244].EXT.BIT19 := FALSE;
   STATUS[244].EXT.BIT20 := FALSE;
   STATUS[244].EXT.AlarmSuppressed := FALSE;
   STATUS[244].EXT.AlarmPresent := FALSE;
   STATUS[244].EXT.AlarmFailUnAck := FALSE;
   STATUS[244].Status := 0;
   STATUS[244].TimeStamp := 16#0000;
   STATUS[245].EXT.AlarmWarnUnAck := FALSE;
   STATUS[245].EXT.AckRequired := FALSE;
   STATUS[245].EXT.Maintanence := FALSE;
   STATUS[245].EXT.Operation := FALSE;
   STATUS[245].EXT.Forced := FALSE;
   STATUS[245].EXT.BIT29 := FALSE;
   STATUS[245].EXT.BIT30 := FALSE;
   STATUS[245].EXT.BIT31 := FALSE;
   STATUS[245].EXT.ModeBit1 := FALSE;
   STATUS[245].EXT.ModeBit2 := FALSE;
   STATUS[245].EXT.ModeBit3 := FALSE;
   STATUS[245].EXT.BIT19 := FALSE;
   STATUS[245].EXT.BIT20 := FALSE;
   STATUS[245].EXT.AlarmSuppressed := FALSE;
   STATUS[245].EXT.AlarmPresent := FALSE;
   STATUS[245].EXT.AlarmFailUnAck := FALSE;
   STATUS[245].Status := 0;
   STATUS[245].TimeStamp := 16#0000;
   STATUS[246].EXT.AlarmWarnUnAck := FALSE;
   STATUS[246].EXT.AckRequired := FALSE;
   STATUS[246].EXT.Maintanence := FALSE;
   STATUS[246].EXT.Operation := FALSE;
   STATUS[246].EXT.Forced := FALSE;
   STATUS[246].EXT.BIT29 := FALSE;
   STATUS[246].EXT.BIT30 := FALSE;
   STATUS[246].EXT.BIT31 := FALSE;
   STATUS[246].EXT.ModeBit1 := FALSE;
   STATUS[246].EXT.ModeBit2 := FALSE;
   STATUS[246].EXT.ModeBit3 := FALSE;
   STATUS[246].EXT.BIT19 := FALSE;
   STATUS[246].EXT.BIT20 := FALSE;
   STATUS[246].EXT.AlarmSuppressed := FALSE;
   STATUS[246].EXT.AlarmPresent := FALSE;
   STATUS[246].EXT.AlarmFailUnAck := FALSE;
   STATUS[246].Status := 0;
   STATUS[246].TimeStamp := 16#0000;
   STATUS[247].EXT.AlarmWarnUnAck := FALSE;
   STATUS[247].EXT.AckRequired := FALSE;
   STATUS[247].EXT.Maintanence := FALSE;
   STATUS[247].EXT.Operation := FALSE;
   STATUS[247].EXT.Forced := FALSE;
   STATUS[247].EXT.BIT29 := FALSE;
   STATUS[247].EXT.BIT30 := FALSE;
   STATUS[247].EXT.BIT31 := FALSE;
   STATUS[247].EXT.ModeBit1 := FALSE;
   STATUS[247].EXT.ModeBit2 := FALSE;
   STATUS[247].EXT.ModeBit3 := FALSE;
   STATUS[247].EXT.BIT19 := FALSE;
   STATUS[247].EXT.BIT20 := FALSE;
   STATUS[247].EXT.AlarmSuppressed := FALSE;
   STATUS[247].EXT.AlarmPresent := FALSE;
   STATUS[247].EXT.AlarmFailUnAck := FALSE;
   STATUS[247].Status := 0;
   STATUS[247].TimeStamp := 16#0000;
   STATUS[248].EXT.AlarmWarnUnAck := FALSE;
   STATUS[248].EXT.AckRequired := FALSE;
   STATUS[248].EXT.Maintanence := FALSE;
   STATUS[248].EXT.Operation := FALSE;
   STATUS[248].EXT.Forced := FALSE;
   STATUS[248].EXT.BIT29 := FALSE;
   STATUS[248].EXT.BIT30 := FALSE;
   STATUS[248].EXT.BIT31 := FALSE;
   STATUS[248].EXT.ModeBit1 := FALSE;
   STATUS[248].EXT.ModeBit2 := FALSE;
   STATUS[248].EXT.ModeBit3 := FALSE;
   STATUS[248].EXT.BIT19 := FALSE;
   STATUS[248].EXT.BIT20 := FALSE;
   STATUS[248].EXT.AlarmSuppressed := FALSE;
   STATUS[248].EXT.AlarmPresent := FALSE;
   STATUS[248].EXT.AlarmFailUnAck := FALSE;
   STATUS[248].Status := 0;
   STATUS[248].TimeStamp := 16#0000;
   STATUS[249].EXT.AlarmWarnUnAck := FALSE;
   STATUS[249].EXT.AckRequired := FALSE;
   STATUS[249].EXT.Maintanence := FALSE;
   STATUS[249].EXT.Operation := FALSE;
   STATUS[249].EXT.Forced := FALSE;
   STATUS[249].EXT.BIT29 := FALSE;
   STATUS[249].EXT.BIT30 := FALSE;
   STATUS[249].EXT.BIT31 := FALSE;
   STATUS[249].EXT.ModeBit1 := FALSE;
   STATUS[249].EXT.ModeBit2 := FALSE;
   STATUS[249].EXT.ModeBit3 := FALSE;
   STATUS[249].EXT.BIT19 := FALSE;
   STATUS[249].EXT.BIT20 := FALSE;
   STATUS[249].EXT.AlarmSuppressed := FALSE;
   STATUS[249].EXT.AlarmPresent := FALSE;
   STATUS[249].EXT.AlarmFailUnAck := FALSE;
   STATUS[249].Status := 0;
   STATUS[249].TimeStamp := 16#0000;
   STATUS[250].EXT.AlarmWarnUnAck := FALSE;
   STATUS[250].EXT.AckRequired := FALSE;
   STATUS[250].EXT.Maintanence := FALSE;
   STATUS[250].EXT.Operation := FALSE;
   STATUS[250].EXT.Forced := FALSE;
   STATUS[250].EXT.BIT29 := FALSE;
   STATUS[250].EXT.BIT30 := FALSE;
   STATUS[250].EXT.BIT31 := FALSE;
   STATUS[250].EXT.ModeBit1 := FALSE;
   STATUS[250].EXT.ModeBit2 := FALSE;
   STATUS[250].EXT.ModeBit3 := FALSE;
   STATUS[250].EXT.BIT19 := FALSE;
   STATUS[250].EXT.BIT20 := FALSE;
   STATUS[250].EXT.AlarmSuppressed := FALSE;
   STATUS[250].EXT.AlarmPresent := FALSE;
   STATUS[250].EXT.AlarmFailUnAck := FALSE;
   STATUS[250].Status := 0;
   STATUS[250].TimeStamp := 16#0000;
   STATUS[251].EXT.AlarmWarnUnAck := FALSE;
   STATUS[251].EXT.AckRequired := FALSE;
   STATUS[251].EXT.Maintanence := FALSE;
   STATUS[251].EXT.Operation := FALSE;
   STATUS[251].EXT.Forced := FALSE;
   STATUS[251].EXT.BIT29 := FALSE;
   STATUS[251].EXT.BIT30 := FALSE;
   STATUS[251].EXT.BIT31 := FALSE;
   STATUS[251].EXT.ModeBit1 := FALSE;
   STATUS[251].EXT.ModeBit2 := FALSE;
   STATUS[251].EXT.ModeBit3 := FALSE;
   STATUS[251].EXT.BIT19 := FALSE;
   STATUS[251].EXT.BIT20 := FALSE;
   STATUS[251].EXT.AlarmSuppressed := FALSE;
   STATUS[251].EXT.AlarmPresent := FALSE;
   STATUS[251].EXT.AlarmFailUnAck := FALSE;
   STATUS[251].Status := 0;
   STATUS[251].TimeStamp := 16#0000;
   STATUS[252].EXT.AlarmWarnUnAck := FALSE;
   STATUS[252].EXT.AckRequired := FALSE;
   STATUS[252].EXT.Maintanence := FALSE;
   STATUS[252].EXT.Operation := FALSE;
   STATUS[252].EXT.Forced := FALSE;
   STATUS[252].EXT.BIT29 := FALSE;
   STATUS[252].EXT.BIT30 := FALSE;
   STATUS[252].EXT.BIT31 := FALSE;
   STATUS[252].EXT.ModeBit1 := FALSE;
   STATUS[252].EXT.ModeBit2 := FALSE;
   STATUS[252].EXT.ModeBit3 := FALSE;
   STATUS[252].EXT.BIT19 := FALSE;
   STATUS[252].EXT.BIT20 := FALSE;
   STATUS[252].EXT.AlarmSuppressed := FALSE;
   STATUS[252].EXT.AlarmPresent := FALSE;
   STATUS[252].EXT.AlarmFailUnAck := FALSE;
   STATUS[252].Status := 0;
   STATUS[252].TimeStamp := 16#0000;
   STATUS[253].EXT.AlarmWarnUnAck := FALSE;
   STATUS[253].EXT.AckRequired := FALSE;
   STATUS[253].EXT.Maintanence := FALSE;
   STATUS[253].EXT.Operation := FALSE;
   STATUS[253].EXT.Forced := FALSE;
   STATUS[253].EXT.BIT29 := FALSE;
   STATUS[253].EXT.BIT30 := FALSE;
   STATUS[253].EXT.BIT31 := FALSE;
   STATUS[253].EXT.ModeBit1 := FALSE;
   STATUS[253].EXT.ModeBit2 := FALSE;
   STATUS[253].EXT.ModeBit3 := FALSE;
   STATUS[253].EXT.BIT19 := FALSE;
   STATUS[253].EXT.BIT20 := FALSE;
   STATUS[253].EXT.AlarmSuppressed := FALSE;
   STATUS[253].EXT.AlarmPresent := FALSE;
   STATUS[253].EXT.AlarmFailUnAck := FALSE;
   STATUS[253].Status := 0;
   STATUS[253].TimeStamp := 16#0000;
   STATUS[254].EXT.AlarmWarnUnAck := FALSE;
   STATUS[254].EXT.AckRequired := FALSE;
   STATUS[254].EXT.Maintanence := FALSE;
   STATUS[254].EXT.Operation := FALSE;
   STATUS[254].EXT.Forced := FALSE;
   STATUS[254].EXT.BIT29 := FALSE;
   STATUS[254].EXT.BIT30 := FALSE;
   STATUS[254].EXT.BIT31 := FALSE;
   STATUS[254].EXT.ModeBit1 := FALSE;
   STATUS[254].EXT.ModeBit2 := FALSE;
   STATUS[254].EXT.ModeBit3 := FALSE;
   STATUS[254].EXT.BIT19 := FALSE;
   STATUS[254].EXT.BIT20 := FALSE;
   STATUS[254].EXT.AlarmSuppressed := FALSE;
   STATUS[254].EXT.AlarmPresent := FALSE;
   STATUS[254].EXT.AlarmFailUnAck := FALSE;
   STATUS[254].Status := 0;
   STATUS[254].TimeStamp := 16#0000;
   STATUS[255].EXT.AlarmWarnUnAck := FALSE;
   STATUS[255].EXT.AckRequired := FALSE;
   STATUS[255].EXT.Maintanence := FALSE;
   STATUS[255].EXT.Operation := FALSE;
   STATUS[255].EXT.Forced := FALSE;
   STATUS[255].EXT.BIT29 := FALSE;
   STATUS[255].EXT.BIT30 := FALSE;
   STATUS[255].EXT.BIT31 := FALSE;
   STATUS[255].EXT.ModeBit1 := FALSE;
   STATUS[255].EXT.ModeBit2 := FALSE;
   STATUS[255].EXT.ModeBit3 := FALSE;
   STATUS[255].EXT.BIT19 := FALSE;
   STATUS[255].EXT.BIT20 := FALSE;
   STATUS[255].EXT.AlarmSuppressed := FALSE;
   STATUS[255].EXT.AlarmPresent := FALSE;
   STATUS[255].EXT.AlarmFailUnAck := FALSE;
   STATUS[255].Status := 0;
   STATUS[255].TimeStamp := 16#0000;
   STATUS[256].EXT.AlarmWarnUnAck := FALSE;
   STATUS[256].EXT.AckRequired := FALSE;
   STATUS[256].EXT.Maintanence := FALSE;
   STATUS[256].EXT.Operation := FALSE;
   STATUS[256].EXT.Forced := FALSE;
   STATUS[256].EXT.BIT29 := FALSE;
   STATUS[256].EXT.BIT30 := FALSE;
   STATUS[256].EXT.BIT31 := FALSE;
   STATUS[256].EXT.ModeBit1 := FALSE;
   STATUS[256].EXT.ModeBit2 := FALSE;
   STATUS[256].EXT.ModeBit3 := FALSE;
   STATUS[256].EXT.BIT19 := FALSE;
   STATUS[256].EXT.BIT20 := FALSE;
   STATUS[256].EXT.AlarmSuppressed := FALSE;
   STATUS[256].EXT.AlarmPresent := FALSE;
   STATUS[256].EXT.AlarmFailUnAck := FALSE;
   STATUS[256].Status := 0;
   STATUS[256].TimeStamp := 16#0000;
   STATUS[257].EXT.AlarmWarnUnAck := FALSE;
   STATUS[257].EXT.AckRequired := FALSE;
   STATUS[257].EXT.Maintanence := FALSE;
   STATUS[257].EXT.Operation := FALSE;
   STATUS[257].EXT.Forced := FALSE;
   STATUS[257].EXT.BIT29 := FALSE;
   STATUS[257].EXT.BIT30 := FALSE;
   STATUS[257].EXT.BIT31 := FALSE;
   STATUS[257].EXT.ModeBit1 := FALSE;
   STATUS[257].EXT.ModeBit2 := FALSE;
   STATUS[257].EXT.ModeBit3 := FALSE;
   STATUS[257].EXT.BIT19 := FALSE;
   STATUS[257].EXT.BIT20 := FALSE;
   STATUS[257].EXT.AlarmSuppressed := FALSE;
   STATUS[257].EXT.AlarmPresent := FALSE;
   STATUS[257].EXT.AlarmFailUnAck := FALSE;
   STATUS[257].Status := 0;
   STATUS[257].TimeStamp := 16#0000;
   STATUS[258].EXT.AlarmWarnUnAck := FALSE;
   STATUS[258].EXT.AckRequired := FALSE;
   STATUS[258].EXT.Maintanence := FALSE;
   STATUS[258].EXT.Operation := FALSE;
   STATUS[258].EXT.Forced := FALSE;
   STATUS[258].EXT.BIT29 := FALSE;
   STATUS[258].EXT.BIT30 := FALSE;
   STATUS[258].EXT.BIT31 := FALSE;
   STATUS[258].EXT.ModeBit1 := FALSE;
   STATUS[258].EXT.ModeBit2 := FALSE;
   STATUS[258].EXT.ModeBit3 := FALSE;
   STATUS[258].EXT.BIT19 := FALSE;
   STATUS[258].EXT.BIT20 := FALSE;
   STATUS[258].EXT.AlarmSuppressed := FALSE;
   STATUS[258].EXT.AlarmPresent := FALSE;
   STATUS[258].EXT.AlarmFailUnAck := FALSE;
   STATUS[258].Status := 0;
   STATUS[258].TimeStamp := 16#0000;
   STATUS[259].EXT.AlarmWarnUnAck := FALSE;
   STATUS[259].EXT.AckRequired := FALSE;
   STATUS[259].EXT.Maintanence := FALSE;
   STATUS[259].EXT.Operation := FALSE;
   STATUS[259].EXT.Forced := FALSE;
   STATUS[259].EXT.BIT29 := FALSE;
   STATUS[259].EXT.BIT30 := FALSE;
   STATUS[259].EXT.BIT31 := FALSE;
   STATUS[259].EXT.ModeBit1 := FALSE;
   STATUS[259].EXT.ModeBit2 := FALSE;
   STATUS[259].EXT.ModeBit3 := FALSE;
   STATUS[259].EXT.BIT19 := FALSE;
   STATUS[259].EXT.BIT20 := FALSE;
   STATUS[259].EXT.AlarmSuppressed := FALSE;
   STATUS[259].EXT.AlarmPresent := FALSE;
   STATUS[259].EXT.AlarmFailUnAck := FALSE;
   STATUS[259].Status := 0;
   STATUS[259].TimeStamp := 16#0000;
   STATUS[260].EXT.AlarmWarnUnAck := FALSE;
   STATUS[260].EXT.AckRequired := FALSE;
   STATUS[260].EXT.Maintanence := FALSE;
   STATUS[260].EXT.Operation := FALSE;
   STATUS[260].EXT.Forced := FALSE;
   STATUS[260].EXT.BIT29 := FALSE;
   STATUS[260].EXT.BIT30 := FALSE;
   STATUS[260].EXT.BIT31 := FALSE;
   STATUS[260].EXT.ModeBit1 := FALSE;
   STATUS[260].EXT.ModeBit2 := FALSE;
   STATUS[260].EXT.ModeBit3 := FALSE;
   STATUS[260].EXT.BIT19 := FALSE;
   STATUS[260].EXT.BIT20 := FALSE;
   STATUS[260].EXT.AlarmSuppressed := FALSE;
   STATUS[260].EXT.AlarmPresent := FALSE;
   STATUS[260].EXT.AlarmFailUnAck := FALSE;
   STATUS[260].Status := 0;
   STATUS[260].TimeStamp := 16#0000;
   STATUS[261].EXT.AlarmWarnUnAck := FALSE;
   STATUS[261].EXT.AckRequired := FALSE;
   STATUS[261].EXT.Maintanence := FALSE;
   STATUS[261].EXT.Operation := FALSE;
   STATUS[261].EXT.Forced := FALSE;
   STATUS[261].EXT.BIT29 := FALSE;
   STATUS[261].EXT.BIT30 := FALSE;
   STATUS[261].EXT.BIT31 := FALSE;
   STATUS[261].EXT.ModeBit1 := FALSE;
   STATUS[261].EXT.ModeBit2 := FALSE;
   STATUS[261].EXT.ModeBit3 := FALSE;
   STATUS[261].EXT.BIT19 := FALSE;
   STATUS[261].EXT.BIT20 := FALSE;
   STATUS[261].EXT.AlarmSuppressed := FALSE;
   STATUS[261].EXT.AlarmPresent := FALSE;
   STATUS[261].EXT.AlarmFailUnAck := FALSE;
   STATUS[261].Status := 0;
   STATUS[261].TimeStamp := 16#0000;
   STATUS[262].EXT.AlarmWarnUnAck := FALSE;
   STATUS[262].EXT.AckRequired := FALSE;
   STATUS[262].EXT.Maintanence := FALSE;
   STATUS[262].EXT.Operation := FALSE;
   STATUS[262].EXT.Forced := FALSE;
   STATUS[262].EXT.BIT29 := FALSE;
   STATUS[262].EXT.BIT30 := FALSE;
   STATUS[262].EXT.BIT31 := FALSE;
   STATUS[262].EXT.ModeBit1 := FALSE;
   STATUS[262].EXT.ModeBit2 := FALSE;
   STATUS[262].EXT.ModeBit3 := FALSE;
   STATUS[262].EXT.BIT19 := FALSE;
   STATUS[262].EXT.BIT20 := FALSE;
   STATUS[262].EXT.AlarmSuppressed := FALSE;
   STATUS[262].EXT.AlarmPresent := FALSE;
   STATUS[262].EXT.AlarmFailUnAck := FALSE;
   STATUS[262].Status := 0;
   STATUS[262].TimeStamp := 16#0000;
   STATUS[263].EXT.AlarmWarnUnAck := FALSE;
   STATUS[263].EXT.AckRequired := FALSE;
   STATUS[263].EXT.Maintanence := FALSE;
   STATUS[263].EXT.Operation := FALSE;
   STATUS[263].EXT.Forced := FALSE;
   STATUS[263].EXT.BIT29 := FALSE;
   STATUS[263].EXT.BIT30 := FALSE;
   STATUS[263].EXT.BIT31 := FALSE;
   STATUS[263].EXT.ModeBit1 := FALSE;
   STATUS[263].EXT.ModeBit2 := FALSE;
   STATUS[263].EXT.ModeBit3 := FALSE;
   STATUS[263].EXT.BIT19 := FALSE;
   STATUS[263].EXT.BIT20 := FALSE;
   STATUS[263].EXT.AlarmSuppressed := FALSE;
   STATUS[263].EXT.AlarmPresent := FALSE;
   STATUS[263].EXT.AlarmFailUnAck := FALSE;
   STATUS[263].Status := 0;
   STATUS[263].TimeStamp := 16#0000;
   STATUS[264].EXT.AlarmWarnUnAck := FALSE;
   STATUS[264].EXT.AckRequired := FALSE;
   STATUS[264].EXT.Maintanence := FALSE;
   STATUS[264].EXT.Operation := FALSE;
   STATUS[264].EXT.Forced := FALSE;
   STATUS[264].EXT.BIT29 := FALSE;
   STATUS[264].EXT.BIT30 := FALSE;
   STATUS[264].EXT.BIT31 := FALSE;
   STATUS[264].EXT.ModeBit1 := FALSE;
   STATUS[264].EXT.ModeBit2 := FALSE;
   STATUS[264].EXT.ModeBit3 := FALSE;
   STATUS[264].EXT.BIT19 := FALSE;
   STATUS[264].EXT.BIT20 := FALSE;
   STATUS[264].EXT.AlarmSuppressed := FALSE;
   STATUS[264].EXT.AlarmPresent := FALSE;
   STATUS[264].EXT.AlarmFailUnAck := FALSE;
   STATUS[264].Status := 0;
   STATUS[264].TimeStamp := 16#0000;
   STATUS[265].EXT.AlarmWarnUnAck := FALSE;
   STATUS[265].EXT.AckRequired := FALSE;
   STATUS[265].EXT.Maintanence := FALSE;
   STATUS[265].EXT.Operation := FALSE;
   STATUS[265].EXT.Forced := FALSE;
   STATUS[265].EXT.BIT29 := FALSE;
   STATUS[265].EXT.BIT30 := FALSE;
   STATUS[265].EXT.BIT31 := FALSE;
   STATUS[265].EXT.ModeBit1 := FALSE;
   STATUS[265].EXT.ModeBit2 := FALSE;
   STATUS[265].EXT.ModeBit3 := FALSE;
   STATUS[265].EXT.BIT19 := FALSE;
   STATUS[265].EXT.BIT20 := FALSE;
   STATUS[265].EXT.AlarmSuppressed := FALSE;
   STATUS[265].EXT.AlarmPresent := FALSE;
   STATUS[265].EXT.AlarmFailUnAck := FALSE;
   STATUS[265].Status := 0;
   STATUS[265].TimeStamp := 16#0000;
   STATUS[266].EXT.AlarmWarnUnAck := FALSE;
   STATUS[266].EXT.AckRequired := FALSE;
   STATUS[266].EXT.Maintanence := FALSE;
   STATUS[266].EXT.Operation := FALSE;
   STATUS[266].EXT.Forced := FALSE;
   STATUS[266].EXT.BIT29 := FALSE;
   STATUS[266].EXT.BIT30 := FALSE;
   STATUS[266].EXT.BIT31 := FALSE;
   STATUS[266].EXT.ModeBit1 := FALSE;
   STATUS[266].EXT.ModeBit2 := FALSE;
   STATUS[266].EXT.ModeBit3 := FALSE;
   STATUS[266].EXT.BIT19 := FALSE;
   STATUS[266].EXT.BIT20 := FALSE;
   STATUS[266].EXT.AlarmSuppressed := FALSE;
   STATUS[266].EXT.AlarmPresent := FALSE;
   STATUS[266].EXT.AlarmFailUnAck := FALSE;
   STATUS[266].Status := 0;
   STATUS[266].TimeStamp := 16#0000;
   STATUS[267].EXT.AlarmWarnUnAck := FALSE;
   STATUS[267].EXT.AckRequired := FALSE;
   STATUS[267].EXT.Maintanence := FALSE;
   STATUS[267].EXT.Operation := FALSE;
   STATUS[267].EXT.Forced := FALSE;
   STATUS[267].EXT.BIT29 := FALSE;
   STATUS[267].EXT.BIT30 := FALSE;
   STATUS[267].EXT.BIT31 := FALSE;
   STATUS[267].EXT.ModeBit1 := FALSE;
   STATUS[267].EXT.ModeBit2 := FALSE;
   STATUS[267].EXT.ModeBit3 := FALSE;
   STATUS[267].EXT.BIT19 := FALSE;
   STATUS[267].EXT.BIT20 := FALSE;
   STATUS[267].EXT.AlarmSuppressed := FALSE;
   STATUS[267].EXT.AlarmPresent := FALSE;
   STATUS[267].EXT.AlarmFailUnAck := FALSE;
   STATUS[267].Status := 0;
   STATUS[267].TimeStamp := 16#0000;
   STATUS[268].EXT.AlarmWarnUnAck := FALSE;
   STATUS[268].EXT.AckRequired := FALSE;
   STATUS[268].EXT.Maintanence := FALSE;
   STATUS[268].EXT.Operation := FALSE;
   STATUS[268].EXT.Forced := FALSE;
   STATUS[268].EXT.BIT29 := FALSE;
   STATUS[268].EXT.BIT30 := FALSE;
   STATUS[268].EXT.BIT31 := FALSE;
   STATUS[268].EXT.ModeBit1 := FALSE;
   STATUS[268].EXT.ModeBit2 := FALSE;
   STATUS[268].EXT.ModeBit3 := FALSE;
   STATUS[268].EXT.BIT19 := FALSE;
   STATUS[268].EXT.BIT20 := FALSE;
   STATUS[268].EXT.AlarmSuppressed := FALSE;
   STATUS[268].EXT.AlarmPresent := FALSE;
   STATUS[268].EXT.AlarmFailUnAck := FALSE;
   STATUS[268].Status := 0;
   STATUS[268].TimeStamp := 16#0000;
   STATUS[269].EXT.AlarmWarnUnAck := FALSE;
   STATUS[269].EXT.AckRequired := FALSE;
   STATUS[269].EXT.Maintanence := FALSE;
   STATUS[269].EXT.Operation := FALSE;
   STATUS[269].EXT.Forced := FALSE;
   STATUS[269].EXT.BIT29 := FALSE;
   STATUS[269].EXT.BIT30 := FALSE;
   STATUS[269].EXT.BIT31 := FALSE;
   STATUS[269].EXT.ModeBit1 := FALSE;
   STATUS[269].EXT.ModeBit2 := FALSE;
   STATUS[269].EXT.ModeBit3 := FALSE;
   STATUS[269].EXT.BIT19 := FALSE;
   STATUS[269].EXT.BIT20 := FALSE;
   STATUS[269].EXT.AlarmSuppressed := FALSE;
   STATUS[269].EXT.AlarmPresent := FALSE;
   STATUS[269].EXT.AlarmFailUnAck := FALSE;
   STATUS[269].Status := 0;
   STATUS[269].TimeStamp := 16#0000;
   STATUS[270].EXT.AlarmWarnUnAck := FALSE;
   STATUS[270].EXT.AckRequired := FALSE;
   STATUS[270].EXT.Maintanence := FALSE;
   STATUS[270].EXT.Operation := FALSE;
   STATUS[270].EXT.Forced := FALSE;
   STATUS[270].EXT.BIT29 := FALSE;
   STATUS[270].EXT.BIT30 := FALSE;
   STATUS[270].EXT.BIT31 := FALSE;
   STATUS[270].EXT.ModeBit1 := FALSE;
   STATUS[270].EXT.ModeBit2 := FALSE;
   STATUS[270].EXT.ModeBit3 := FALSE;
   STATUS[270].EXT.BIT19 := FALSE;
   STATUS[270].EXT.BIT20 := FALSE;
   STATUS[270].EXT.AlarmSuppressed := FALSE;
   STATUS[270].EXT.AlarmPresent := FALSE;
   STATUS[270].EXT.AlarmFailUnAck := FALSE;
   STATUS[270].Status := 0;
   STATUS[270].TimeStamp := 16#0000;
   STATUS[271].EXT.AlarmWarnUnAck := FALSE;
   STATUS[271].EXT.AckRequired := FALSE;
   STATUS[271].EXT.Maintanence := FALSE;
   STATUS[271].EXT.Operation := FALSE;
   STATUS[271].EXT.Forced := FALSE;
   STATUS[271].EXT.BIT29 := FALSE;
   STATUS[271].EXT.BIT30 := FALSE;
   STATUS[271].EXT.BIT31 := FALSE;
   STATUS[271].EXT.ModeBit1 := FALSE;
   STATUS[271].EXT.ModeBit2 := FALSE;
   STATUS[271].EXT.ModeBit3 := FALSE;
   STATUS[271].EXT.BIT19 := FALSE;
   STATUS[271].EXT.BIT20 := FALSE;
   STATUS[271].EXT.AlarmSuppressed := FALSE;
   STATUS[271].EXT.AlarmPresent := FALSE;
   STATUS[271].EXT.AlarmFailUnAck := FALSE;
   STATUS[271].Status := 0;
   STATUS[271].TimeStamp := 16#0000;
   STATUS[272].EXT.AlarmWarnUnAck := FALSE;
   STATUS[272].EXT.AckRequired := FALSE;
   STATUS[272].EXT.Maintanence := FALSE;
   STATUS[272].EXT.Operation := FALSE;
   STATUS[272].EXT.Forced := FALSE;
   STATUS[272].EXT.BIT29 := FALSE;
   STATUS[272].EXT.BIT30 := FALSE;
   STATUS[272].EXT.BIT31 := FALSE;
   STATUS[272].EXT.ModeBit1 := FALSE;
   STATUS[272].EXT.ModeBit2 := FALSE;
   STATUS[272].EXT.ModeBit3 := FALSE;
   STATUS[272].EXT.BIT19 := FALSE;
   STATUS[272].EXT.BIT20 := FALSE;
   STATUS[272].EXT.AlarmSuppressed := FALSE;
   STATUS[272].EXT.AlarmPresent := FALSE;
   STATUS[272].EXT.AlarmFailUnAck := FALSE;
   STATUS[272].Status := 0;
   STATUS[272].TimeStamp := 16#0000;
   STATUS[273].EXT.AlarmWarnUnAck := FALSE;
   STATUS[273].EXT.AckRequired := FALSE;
   STATUS[273].EXT.Maintanence := FALSE;
   STATUS[273].EXT.Operation := FALSE;
   STATUS[273].EXT.Forced := FALSE;
   STATUS[273].EXT.BIT29 := FALSE;
   STATUS[273].EXT.BIT30 := FALSE;
   STATUS[273].EXT.BIT31 := FALSE;
   STATUS[273].EXT.ModeBit1 := FALSE;
   STATUS[273].EXT.ModeBit2 := FALSE;
   STATUS[273].EXT.ModeBit3 := FALSE;
   STATUS[273].EXT.BIT19 := FALSE;
   STATUS[273].EXT.BIT20 := FALSE;
   STATUS[273].EXT.AlarmSuppressed := FALSE;
   STATUS[273].EXT.AlarmPresent := FALSE;
   STATUS[273].EXT.AlarmFailUnAck := FALSE;
   STATUS[273].Status := 0;
   STATUS[273].TimeStamp := 16#0000;
   STATUS[274].EXT.AlarmWarnUnAck := FALSE;
   STATUS[274].EXT.AckRequired := FALSE;
   STATUS[274].EXT.Maintanence := FALSE;
   STATUS[274].EXT.Operation := FALSE;
   STATUS[274].EXT.Forced := FALSE;
   STATUS[274].EXT.BIT29 := FALSE;
   STATUS[274].EXT.BIT30 := FALSE;
   STATUS[274].EXT.BIT31 := FALSE;
   STATUS[274].EXT.ModeBit1 := FALSE;
   STATUS[274].EXT.ModeBit2 := FALSE;
   STATUS[274].EXT.ModeBit3 := FALSE;
   STATUS[274].EXT.BIT19 := FALSE;
   STATUS[274].EXT.BIT20 := FALSE;
   STATUS[274].EXT.AlarmSuppressed := FALSE;
   STATUS[274].EXT.AlarmPresent := FALSE;
   STATUS[274].EXT.AlarmFailUnAck := FALSE;
   STATUS[274].Status := 0;
   STATUS[274].TimeStamp := 16#0000;
   STATUS[275].EXT.AlarmWarnUnAck := FALSE;
   STATUS[275].EXT.AckRequired := FALSE;
   STATUS[275].EXT.Maintanence := FALSE;
   STATUS[275].EXT.Operation := FALSE;
   STATUS[275].EXT.Forced := FALSE;
   STATUS[275].EXT.BIT29 := FALSE;
   STATUS[275].EXT.BIT30 := FALSE;
   STATUS[275].EXT.BIT31 := FALSE;
   STATUS[275].EXT.ModeBit1 := FALSE;
   STATUS[275].EXT.ModeBit2 := FALSE;
   STATUS[275].EXT.ModeBit3 := FALSE;
   STATUS[275].EXT.BIT19 := FALSE;
   STATUS[275].EXT.BIT20 := FALSE;
   STATUS[275].EXT.AlarmSuppressed := FALSE;
   STATUS[275].EXT.AlarmPresent := FALSE;
   STATUS[275].EXT.AlarmFailUnAck := FALSE;
   STATUS[275].Status := 0;
   STATUS[275].TimeStamp := 16#0000;
   STATUS[276].EXT.AlarmWarnUnAck := FALSE;
   STATUS[276].EXT.AckRequired := FALSE;
   STATUS[276].EXT.Maintanence := FALSE;
   STATUS[276].EXT.Operation := FALSE;
   STATUS[276].EXT.Forced := FALSE;
   STATUS[276].EXT.BIT29 := FALSE;
   STATUS[276].EXT.BIT30 := FALSE;
   STATUS[276].EXT.BIT31 := FALSE;
   STATUS[276].EXT.ModeBit1 := FALSE;
   STATUS[276].EXT.ModeBit2 := FALSE;
   STATUS[276].EXT.ModeBit3 := FALSE;
   STATUS[276].EXT.BIT19 := FALSE;
   STATUS[276].EXT.BIT20 := FALSE;
   STATUS[276].EXT.AlarmSuppressed := FALSE;
   STATUS[276].EXT.AlarmPresent := FALSE;
   STATUS[276].EXT.AlarmFailUnAck := FALSE;
   STATUS[276].Status := 0;
   STATUS[276].TimeStamp := 16#0000;
   STATUS[277].EXT.AlarmWarnUnAck := FALSE;
   STATUS[277].EXT.AckRequired := FALSE;
   STATUS[277].EXT.Maintanence := FALSE;
   STATUS[277].EXT.Operation := FALSE;
   STATUS[277].EXT.Forced := FALSE;
   STATUS[277].EXT.BIT29 := FALSE;
   STATUS[277].EXT.BIT30 := FALSE;
   STATUS[277].EXT.BIT31 := FALSE;
   STATUS[277].EXT.ModeBit1 := FALSE;
   STATUS[277].EXT.ModeBit2 := FALSE;
   STATUS[277].EXT.ModeBit3 := FALSE;
   STATUS[277].EXT.BIT19 := FALSE;
   STATUS[277].EXT.BIT20 := FALSE;
   STATUS[277].EXT.AlarmSuppressed := FALSE;
   STATUS[277].EXT.AlarmPresent := FALSE;
   STATUS[277].EXT.AlarmFailUnAck := FALSE;
   STATUS[277].Status := 0;
   STATUS[277].TimeStamp := 16#0000;
   STATUS[278].EXT.AlarmWarnUnAck := FALSE;
   STATUS[278].EXT.AckRequired := FALSE;
   STATUS[278].EXT.Maintanence := FALSE;
   STATUS[278].EXT.Operation := FALSE;
   STATUS[278].EXT.Forced := FALSE;
   STATUS[278].EXT.BIT29 := FALSE;
   STATUS[278].EXT.BIT30 := FALSE;
   STATUS[278].EXT.BIT31 := FALSE;
   STATUS[278].EXT.ModeBit1 := FALSE;
   STATUS[278].EXT.ModeBit2 := FALSE;
   STATUS[278].EXT.ModeBit3 := FALSE;
   STATUS[278].EXT.BIT19 := FALSE;
   STATUS[278].EXT.BIT20 := FALSE;
   STATUS[278].EXT.AlarmSuppressed := FALSE;
   STATUS[278].EXT.AlarmPresent := FALSE;
   STATUS[278].EXT.AlarmFailUnAck := FALSE;
   STATUS[278].Status := 0;
   STATUS[278].TimeStamp := 16#0000;
   STATUS[279].EXT.AlarmWarnUnAck := FALSE;
   STATUS[279].EXT.AckRequired := FALSE;
   STATUS[279].EXT.Maintanence := FALSE;
   STATUS[279].EXT.Operation := FALSE;
   STATUS[279].EXT.Forced := FALSE;
   STATUS[279].EXT.BIT29 := FALSE;
   STATUS[279].EXT.BIT30 := FALSE;
   STATUS[279].EXT.BIT31 := FALSE;
   STATUS[279].EXT.ModeBit1 := FALSE;
   STATUS[279].EXT.ModeBit2 := FALSE;
   STATUS[279].EXT.ModeBit3 := FALSE;
   STATUS[279].EXT.BIT19 := FALSE;
   STATUS[279].EXT.BIT20 := FALSE;
   STATUS[279].EXT.AlarmSuppressed := FALSE;
   STATUS[279].EXT.AlarmPresent := FALSE;
   STATUS[279].EXT.AlarmFailUnAck := FALSE;
   STATUS[279].Status := 0;
   STATUS[279].TimeStamp := 16#0000;
   STATUS[280].EXT.AlarmWarnUnAck := FALSE;
   STATUS[280].EXT.AckRequired := FALSE;
   STATUS[280].EXT.Maintanence := FALSE;
   STATUS[280].EXT.Operation := FALSE;
   STATUS[280].EXT.Forced := FALSE;
   STATUS[280].EXT.BIT29 := FALSE;
   STATUS[280].EXT.BIT30 := FALSE;
   STATUS[280].EXT.BIT31 := FALSE;
   STATUS[280].EXT.ModeBit1 := FALSE;
   STATUS[280].EXT.ModeBit2 := FALSE;
   STATUS[280].EXT.ModeBit3 := FALSE;
   STATUS[280].EXT.BIT19 := FALSE;
   STATUS[280].EXT.BIT20 := FALSE;
   STATUS[280].EXT.AlarmSuppressed := FALSE;
   STATUS[280].EXT.AlarmPresent := FALSE;
   STATUS[280].EXT.AlarmFailUnAck := FALSE;
   STATUS[280].Status := 0;
   STATUS[280].TimeStamp := 16#0000;
   STATUS[281].EXT.AlarmWarnUnAck := FALSE;
   STATUS[281].EXT.AckRequired := FALSE;
   STATUS[281].EXT.Maintanence := FALSE;
   STATUS[281].EXT.Operation := FALSE;
   STATUS[281].EXT.Forced := FALSE;
   STATUS[281].EXT.BIT29 := FALSE;
   STATUS[281].EXT.BIT30 := FALSE;
   STATUS[281].EXT.BIT31 := FALSE;
   STATUS[281].EXT.ModeBit1 := FALSE;
   STATUS[281].EXT.ModeBit2 := FALSE;
   STATUS[281].EXT.ModeBit3 := FALSE;
   STATUS[281].EXT.BIT19 := FALSE;
   STATUS[281].EXT.BIT20 := FALSE;
   STATUS[281].EXT.AlarmSuppressed := FALSE;
   STATUS[281].EXT.AlarmPresent := FALSE;
   STATUS[281].EXT.AlarmFailUnAck := FALSE;
   STATUS[281].Status := 0;
   STATUS[281].TimeStamp := 16#0000;
   STATUS[282].EXT.AlarmWarnUnAck := FALSE;
   STATUS[282].EXT.AckRequired := FALSE;
   STATUS[282].EXT.Maintanence := FALSE;
   STATUS[282].EXT.Operation := FALSE;
   STATUS[282].EXT.Forced := FALSE;
   STATUS[282].EXT.BIT29 := FALSE;
   STATUS[282].EXT.BIT30 := FALSE;
   STATUS[282].EXT.BIT31 := FALSE;
   STATUS[282].EXT.ModeBit1 := FALSE;
   STATUS[282].EXT.ModeBit2 := FALSE;
   STATUS[282].EXT.ModeBit3 := FALSE;
   STATUS[282].EXT.BIT19 := FALSE;
   STATUS[282].EXT.BIT20 := FALSE;
   STATUS[282].EXT.AlarmSuppressed := FALSE;
   STATUS[282].EXT.AlarmPresent := FALSE;
   STATUS[282].EXT.AlarmFailUnAck := FALSE;
   STATUS[282].Status := 0;
   STATUS[282].TimeStamp := 16#0000;
   STATUS[283].EXT.AlarmWarnUnAck := FALSE;
   STATUS[283].EXT.AckRequired := FALSE;
   STATUS[283].EXT.Maintanence := FALSE;
   STATUS[283].EXT.Operation := FALSE;
   STATUS[283].EXT.Forced := FALSE;
   STATUS[283].EXT.BIT29 := FALSE;
   STATUS[283].EXT.BIT30 := FALSE;
   STATUS[283].EXT.BIT31 := FALSE;
   STATUS[283].EXT.ModeBit1 := FALSE;
   STATUS[283].EXT.ModeBit2 := FALSE;
   STATUS[283].EXT.ModeBit3 := FALSE;
   STATUS[283].EXT.BIT19 := FALSE;
   STATUS[283].EXT.BIT20 := FALSE;
   STATUS[283].EXT.AlarmSuppressed := FALSE;
   STATUS[283].EXT.AlarmPresent := FALSE;
   STATUS[283].EXT.AlarmFailUnAck := FALSE;
   STATUS[283].Status := 0;
   STATUS[283].TimeStamp := 16#0000;
   STATUS[284].EXT.AlarmWarnUnAck := FALSE;
   STATUS[284].EXT.AckRequired := FALSE;
   STATUS[284].EXT.Maintanence := FALSE;
   STATUS[284].EXT.Operation := FALSE;
   STATUS[284].EXT.Forced := FALSE;
   STATUS[284].EXT.BIT29 := FALSE;
   STATUS[284].EXT.BIT30 := FALSE;
   STATUS[284].EXT.BIT31 := FALSE;
   STATUS[284].EXT.ModeBit1 := FALSE;
   STATUS[284].EXT.ModeBit2 := FALSE;
   STATUS[284].EXT.ModeBit3 := FALSE;
   STATUS[284].EXT.BIT19 := FALSE;
   STATUS[284].EXT.BIT20 := FALSE;
   STATUS[284].EXT.AlarmSuppressed := FALSE;
   STATUS[284].EXT.AlarmPresent := FALSE;
   STATUS[284].EXT.AlarmFailUnAck := FALSE;
   STATUS[284].Status := 0;
   STATUS[284].TimeStamp := 16#0000;
   STATUS[285].EXT.AlarmWarnUnAck := FALSE;
   STATUS[285].EXT.AckRequired := FALSE;
   STATUS[285].EXT.Maintanence := FALSE;
   STATUS[285].EXT.Operation := FALSE;
   STATUS[285].EXT.Forced := FALSE;
   STATUS[285].EXT.BIT29 := FALSE;
   STATUS[285].EXT.BIT30 := FALSE;
   STATUS[285].EXT.BIT31 := FALSE;
   STATUS[285].EXT.ModeBit1 := FALSE;
   STATUS[285].EXT.ModeBit2 := FALSE;
   STATUS[285].EXT.ModeBit3 := FALSE;
   STATUS[285].EXT.BIT19 := FALSE;
   STATUS[285].EXT.BIT20 := FALSE;
   STATUS[285].EXT.AlarmSuppressed := FALSE;
   STATUS[285].EXT.AlarmPresent := FALSE;
   STATUS[285].EXT.AlarmFailUnAck := FALSE;
   STATUS[285].Status := 0;
   STATUS[285].TimeStamp := 16#0000;
   STATUS[286].EXT.AlarmWarnUnAck := FALSE;
   STATUS[286].EXT.AckRequired := FALSE;
   STATUS[286].EXT.Maintanence := FALSE;
   STATUS[286].EXT.Operation := FALSE;
   STATUS[286].EXT.Forced := FALSE;
   STATUS[286].EXT.BIT29 := FALSE;
   STATUS[286].EXT.BIT30 := FALSE;
   STATUS[286].EXT.BIT31 := FALSE;
   STATUS[286].EXT.ModeBit1 := FALSE;
   STATUS[286].EXT.ModeBit2 := FALSE;
   STATUS[286].EXT.ModeBit3 := FALSE;
   STATUS[286].EXT.BIT19 := FALSE;
   STATUS[286].EXT.BIT20 := FALSE;
   STATUS[286].EXT.AlarmSuppressed := FALSE;
   STATUS[286].EXT.AlarmPresent := FALSE;
   STATUS[286].EXT.AlarmFailUnAck := FALSE;
   STATUS[286].Status := 0;
   STATUS[286].TimeStamp := 16#0000;
   STATUS[287].EXT.AlarmWarnUnAck := FALSE;
   STATUS[287].EXT.AckRequired := FALSE;
   STATUS[287].EXT.Maintanence := FALSE;
   STATUS[287].EXT.Operation := FALSE;
   STATUS[287].EXT.Forced := FALSE;
   STATUS[287].EXT.BIT29 := FALSE;
   STATUS[287].EXT.BIT30 := FALSE;
   STATUS[287].EXT.BIT31 := FALSE;
   STATUS[287].EXT.ModeBit1 := FALSE;
   STATUS[287].EXT.ModeBit2 := FALSE;
   STATUS[287].EXT.ModeBit3 := FALSE;
   STATUS[287].EXT.BIT19 := FALSE;
   STATUS[287].EXT.BIT20 := FALSE;
   STATUS[287].EXT.AlarmSuppressed := FALSE;
   STATUS[287].EXT.AlarmPresent := FALSE;
   STATUS[287].EXT.AlarmFailUnAck := FALSE;
   STATUS[287].Status := 0;
   STATUS[287].TimeStamp := 16#0000;
   STATUS[288].EXT.AlarmWarnUnAck := FALSE;
   STATUS[288].EXT.AckRequired := FALSE;
   STATUS[288].EXT.Maintanence := FALSE;
   STATUS[288].EXT.Operation := FALSE;
   STATUS[288].EXT.Forced := FALSE;
   STATUS[288].EXT.BIT29 := FALSE;
   STATUS[288].EXT.BIT30 := FALSE;
   STATUS[288].EXT.BIT31 := FALSE;
   STATUS[288].EXT.ModeBit1 := FALSE;
   STATUS[288].EXT.ModeBit2 := FALSE;
   STATUS[288].EXT.ModeBit3 := FALSE;
   STATUS[288].EXT.BIT19 := FALSE;
   STATUS[288].EXT.BIT20 := FALSE;
   STATUS[288].EXT.AlarmSuppressed := FALSE;
   STATUS[288].EXT.AlarmPresent := FALSE;
   STATUS[288].EXT.AlarmFailUnAck := FALSE;
   STATUS[288].Status := 0;
   STATUS[288].TimeStamp := 16#0000;
   STATUS[289].EXT.AlarmWarnUnAck := FALSE;
   STATUS[289].EXT.AckRequired := FALSE;
   STATUS[289].EXT.Maintanence := FALSE;
   STATUS[289].EXT.Operation := FALSE;
   STATUS[289].EXT.Forced := FALSE;
   STATUS[289].EXT.BIT29 := FALSE;
   STATUS[289].EXT.BIT30 := FALSE;
   STATUS[289].EXT.BIT31 := FALSE;
   STATUS[289].EXT.ModeBit1 := FALSE;
   STATUS[289].EXT.ModeBit2 := FALSE;
   STATUS[289].EXT.ModeBit3 := FALSE;
   STATUS[289].EXT.BIT19 := FALSE;
   STATUS[289].EXT.BIT20 := FALSE;
   STATUS[289].EXT.AlarmSuppressed := FALSE;
   STATUS[289].EXT.AlarmPresent := FALSE;
   STATUS[289].EXT.AlarmFailUnAck := FALSE;
   STATUS[289].Status := 0;
   STATUS[289].TimeStamp := 16#0000;
   STATUS[290].EXT.AlarmWarnUnAck := FALSE;
   STATUS[290].EXT.AckRequired := FALSE;
   STATUS[290].EXT.Maintanence := FALSE;
   STATUS[290].EXT.Operation := FALSE;
   STATUS[290].EXT.Forced := FALSE;
   STATUS[290].EXT.BIT29 := FALSE;
   STATUS[290].EXT.BIT30 := FALSE;
   STATUS[290].EXT.BIT31 := FALSE;
   STATUS[290].EXT.ModeBit1 := FALSE;
   STATUS[290].EXT.ModeBit2 := FALSE;
   STATUS[290].EXT.ModeBit3 := FALSE;
   STATUS[290].EXT.BIT19 := FALSE;
   STATUS[290].EXT.BIT20 := FALSE;
   STATUS[290].EXT.AlarmSuppressed := FALSE;
   STATUS[290].EXT.AlarmPresent := FALSE;
   STATUS[290].EXT.AlarmFailUnAck := FALSE;
   STATUS[290].Status := 0;
   STATUS[290].TimeStamp := 16#0000;
   STATUS[291].EXT.AlarmWarnUnAck := FALSE;
   STATUS[291].EXT.AckRequired := FALSE;
   STATUS[291].EXT.Maintanence := FALSE;
   STATUS[291].EXT.Operation := FALSE;
   STATUS[291].EXT.Forced := FALSE;
   STATUS[291].EXT.BIT29 := FALSE;
   STATUS[291].EXT.BIT30 := FALSE;
   STATUS[291].EXT.BIT31 := FALSE;
   STATUS[291].EXT.ModeBit1 := FALSE;
   STATUS[291].EXT.ModeBit2 := FALSE;
   STATUS[291].EXT.ModeBit3 := FALSE;
   STATUS[291].EXT.BIT19 := FALSE;
   STATUS[291].EXT.BIT20 := FALSE;
   STATUS[291].EXT.AlarmSuppressed := FALSE;
   STATUS[291].EXT.AlarmPresent := FALSE;
   STATUS[291].EXT.AlarmFailUnAck := FALSE;
   STATUS[291].Status := 0;
   STATUS[291].TimeStamp := 16#0000;
   STATUS[292].EXT.AlarmWarnUnAck := FALSE;
   STATUS[292].EXT.AckRequired := FALSE;
   STATUS[292].EXT.Maintanence := FALSE;
   STATUS[292].EXT.Operation := FALSE;
   STATUS[292].EXT.Forced := FALSE;
   STATUS[292].EXT.BIT29 := FALSE;
   STATUS[292].EXT.BIT30 := FALSE;
   STATUS[292].EXT.BIT31 := FALSE;
   STATUS[292].EXT.ModeBit1 := FALSE;
   STATUS[292].EXT.ModeBit2 := FALSE;
   STATUS[292].EXT.ModeBit3 := FALSE;
   STATUS[292].EXT.BIT19 := FALSE;
   STATUS[292].EXT.BIT20 := FALSE;
   STATUS[292].EXT.AlarmSuppressed := FALSE;
   STATUS[292].EXT.AlarmPresent := FALSE;
   STATUS[292].EXT.AlarmFailUnAck := FALSE;
   STATUS[292].Status := 0;
   STATUS[292].TimeStamp := 16#0000;
   STATUS[293].EXT.AlarmWarnUnAck := FALSE;
   STATUS[293].EXT.AckRequired := FALSE;
   STATUS[293].EXT.Maintanence := FALSE;
   STATUS[293].EXT.Operation := FALSE;
   STATUS[293].EXT.Forced := FALSE;
   STATUS[293].EXT.BIT29 := FALSE;
   STATUS[293].EXT.BIT30 := FALSE;
   STATUS[293].EXT.BIT31 := FALSE;
   STATUS[293].EXT.ModeBit1 := FALSE;
   STATUS[293].EXT.ModeBit2 := FALSE;
   STATUS[293].EXT.ModeBit3 := FALSE;
   STATUS[293].EXT.BIT19 := FALSE;
   STATUS[293].EXT.BIT20 := FALSE;
   STATUS[293].EXT.AlarmSuppressed := FALSE;
   STATUS[293].EXT.AlarmPresent := FALSE;
   STATUS[293].EXT.AlarmFailUnAck := FALSE;
   STATUS[293].Status := 0;
